Omron Sysmac Studio project 15-510_8110_20151007_10 (Sysmac Studio 1.1.4.95, StandardProject)

# Controller S8130_8140: NJ101-1000 version 1.10
Task PrimaryTask (priority 4, period or condition 1000): Program0, Program1, Program2, prS8120CCD

TYPE WORD_UNION : UNION
    Word_Type : WORD;
    Byte_Type : ARRAY[0..1] OF BYTE;
    Bool_Type : ARRAY[0..15] OF BOOL;
END_UNION END_TYPE
TYPE WorkType : STRUCT
    CCDSectionNo : INT;
    MotionData : Postion;
    QuantityofScrew : ARRAY[0..2] OF ScrewQuantity;
END_STRUCT END_TYPE
TYPE Postion : STRUCT
    Address : DINT;
    Speed : DINT;
END_STRUCT END_TYPE
TYPE ScrewQuantity : STRUCT
    Quantity : INT;
    ScrewJobNo : INT;
END_STRUCT END_TYPE
TYPE RecordData : STRUCT
    WorkingFlag : BOOL;
    FinishFlag : BOOL;
    OKFlag : BOOL;
    NGFlag : BOOL;
END_STRUCT END_TYPE
TYPE FH_CommandCode : (ChangeType := 3149824); END_TYPE

VAR_GLOBAL
    Reset_PB : BOOL;  (* 復歸開關; at IOBus://rack#0/slot#0/Ch1_In/Ch1_In00 *)
    EStop_PB : BOOL;  (* 急停開關; at IOBus://rack#0/slot#0/Ch1_In/Ch1_In01 *)
    CCDStart_PB : BOOL;  (* CCD啟動開關; at IOBus://rack#0/slot#0/Ch1_In/Ch1_In02 *)
    NGReject_SNR : BOOL;  (* 不良品排除檢測; at IOBus://rack#0/slot#0/Ch1_In/Ch1_In03 *)
    S8120_OK : BOOL;  (* at IOBus://rack#0/slot#0/Ch1_In/Ch1_In04 *)
    S8120_NG : BOOL;  (* at IOBus://rack#0/slot#0/Ch1_In/Ch1_In05 *)
    ASDA_IN_SRDY : BOOL;  (* at IOBus://rack#0/slot#0/Ch1_In/Ch1_In06 *)
    ASDA_IN_ZSPD : BOOL;  (* at IOBus://rack#0/slot#0/Ch1_In/Ch1_In07 *)
    ASDA_IN_HOME : BOOL;  (* at IOBus://rack#0/slot#0/Ch1_In/Ch1_In08 *)
    FeedScrew1_FeedSol : BOOL;  (* 送螺絲節流電磁閥1; at IOBus://rack#0/slot#0/Ch1_In/Ch1_In10 *)
    FeedScrew1_FeedSNR : BOOL;  (* 送螺絲螺絲檢知1; at IOBus://rack#0/slot#0/Ch1_In/Ch1_In11 *)
    FeedScrew2_FeedSol : BOOL;  (* 送螺絲節流電磁閥2; at IOBus://rack#0/slot#0/Ch1_In/Ch1_In12 *)
    FeedScrew2_FeedSNR : BOOL;  (* 送螺絲螺絲檢知2; at IOBus://rack#0/slot#0/Ch1_In/Ch1_In13 *)
    FeedScrew3_FeedSol : BOOL;  (* 送螺絲節流電磁閥3; at IOBus://rack#0/slot#0/Ch1_In/Ch1_In14 *)
    FeedScrew3_FeedSNR : BOOL;  (* 送螺絲螺絲檢知3; at IOBus://rack#0/slot#0/Ch1_In/Ch1_In15 *)
    Stanley1_IN_InCycle : BOOL;  (* 鎖付伺服左; at IOBus://rack#0/slot#0/Ch2_In/Ch2_In00 *)
    Stanley1_IN_Ready : BOOL;  (* 鎖付伺服左; at IOBus://rack#0/slot#0/Ch2_In/Ch2_In01 *)
    Stanley1_IN_DisassemblyDetected : BOOL;  (* 鎖付伺服左; at IOBus://rack#0/slot#0/Ch2_In/Ch2_In02 *)
    Stanley1_IN_JobSelectedBit0 : BOOL;  (* 鎖付伺服左; at IOBus://rack#0/slot#0/Ch2_In/Ch2_In03 *)
    Stanley1_IN_JobSelectedBit1 : BOOL;  (* 鎖付伺服左; at IOBus://rack#0/slot#0/Ch2_In/Ch2_In04 *)
    Stanley1_IN_JobSelectedBit2 : BOOL;  (* 鎖付伺服左; at IOBus://rack#0/slot#0/Ch2_In/Ch2_In05 *)
    Stanley1_IN_CycleOK : BOOL;  (* 鎖付伺服左; at IOBus://rack#0/slot#0/Ch2_In/Ch2_In06 *)
    Stanley1_IN_CycleNOK : BOOL;  (* 鎖付伺服左; at IOBus://rack#0/slot#0/Ch2_In/Ch2_In07 *)
    Stanley2_IN_InCycle : BOOL;  (* 鎖付伺服右; at IOBus://rack#0/slot#0/Ch2_In/Ch2_In08 *)
    Stanley2_IN_Ready : BOOL;  (* 鎖付伺服右; at IOBus://rack#0/slot#0/Ch2_In/Ch2_In09 *)
    Stanley2_IN_DisassemblyDetected : BOOL;  (* 鎖付伺服右; at IOBus://rack#0/slot#0/Ch2_In/Ch2_In10 *)
    Stanley2_IN_JobSelectedBit0 : BOOL;  (* 鎖付伺服右; at IOBus://rack#0/slot#0/Ch2_In/Ch2_In11 *)
    Stanley2_IN_JobSelectedBit1 : BOOL;  (* 鎖付伺服右; at IOBus://rack#0/slot#0/Ch2_In/Ch2_In12 *)
    Stanley2_IN_JobSelectedBit2 : BOOL;  (* 鎖付伺服右; at IOBus://rack#0/slot#0/Ch2_In/Ch2_In13 *)
    Stanley2_IN_CycleOK : BOOL;  (* 鎖付伺服右; at IOBus://rack#0/slot#0/Ch2_In/Ch2_In14 *)
    Stanley2_IN_CycleNOK : BOOL;  (* 鎖付伺服右; at IOBus://rack#0/slot#0/Ch2_In/Ch2_In15 *)
    FeedScrew1_FeedRY : BOOL;  (* 送螺絲啟動_1; at IOBus://rack#0/slot#1/Ch1_Out/Ch1_Out00 *)
    FeedScrew2_FeedRY : BOOL;  (* 送螺絲啟動_2; at IOBus://rack#0/slot#1/Ch1_Out/Ch1_Out01 *)
    FeedScrew3_FeedRY : BOOL;  (* 送螺絲啟動_3; at IOBus://rack#0/slot#1/Ch1_Out/Ch1_Out02 *)
    BZ : BOOL;  (* 蜂鳴器; at IOBus://rack#0/slot#1/Ch1_Out/Ch1_Out04 *)
    YL : BOOL;  (* 黃燈; at IOBus://rack#0/slot#1/Ch1_Out/Ch1_Out05 *)
    GL : BOOL;  (* 綠燈; at IOBus://rack#0/slot#1/Ch1_Out/Ch1_Out06 *)
    RL : BOOL;  (* 紅燈; at IOBus://rack#0/slot#1/Ch1_Out/Ch1_Out07 *)
    ASDA_OUT_ARST : BOOL;  (* at IOBus://rack#0/slot#1/Ch1_Out/Ch1_Out11 *)
    Stanley1_OUT_Start : BOOL;  (* 鎖付伺服左; at IOBus://rack#0/slot#1/Ch2_Out/Ch2_Out00 *)
    Stanley1_OUT_Stop : BOOL;  (* 鎖付伺服左; at IOBus://rack#0/slot#1/Ch2_Out/Ch2_Out01 *)
    Stanley1_OUT_Reverse : BOOL;  (* 鎖付伺服左; at IOBus://rack#0/slot#1/Ch2_Out/Ch2_Out02 *)
    Stanley1_OUT_JobBit0 : BOOL;  (* 鎖付伺服左; at IOBus://rack#0/slot#1/Ch2_Out/Ch2_Out03 *)
    Stanley1_OUT_JobBit1 : BOOL;  (* 鎖付伺服左; at IOBus://rack#0/slot#1/Ch2_Out/Ch2_Out04 *)
    Stanley1_OUT_JobBit2 : BOOL;  (* 鎖付伺服左; at IOBus://rack#0/slot#1/Ch2_Out/Ch2_Out05 *)
    Stanley1_OUT_RsetJob : BOOL;  (* 鎖付伺服左; at IOBus://rack#0/slot#1/Ch2_Out/Ch2_Out06 *)
    Stanley1_OUT_Ignored : BOOL;  (* 鎖付伺服左; at IOBus://rack#0/slot#1/Ch2_Out/Ch2_Out07 *)
    Stanley2_OUT_Start : BOOL;  (* 鎖付伺服右; at IOBus://rack#0/slot#1/Ch2_Out/Ch2_Out08 *)
    Stanley2_OUT_Stop : BOOL;  (* 鎖付伺服右; at IOBus://rack#0/slot#1/Ch2_Out/Ch2_Out09 *)
    Stanley2_OUT_Reverse : BOOL;  (* 鎖付伺服右; at IOBus://rack#0/slot#1/Ch2_Out/Ch2_Out10 *)
    Stanley2_OUT_JobBit0 : BOOL;  (* 鎖付伺服右; at IOBus://rack#0/slot#1/Ch2_Out/Ch2_Out11 *)
    Stanley2_OUT_JobBit1 : BOOL;  (* 鎖付伺服右; at IOBus://rack#0/slot#1/Ch2_Out/Ch2_Out12 *)
    Stanley2_OUT_JobBit2 : BOOL;  (* 鎖付伺服右; at IOBus://rack#0/slot#1/Ch2_Out/Ch2_Out13 *)
    Stanley2_OUT_RsetJob : BOOL;  (* 鎖付伺服右; at IOBus://rack#0/slot#1/Ch2_Out/Ch2_Out14 *)
    Stanley2_OUT_Ignored : BOOL;  (* 鎖付伺服右; at IOBus://rack#0/slot#1/Ch2_Out/Ch2_Out15 *)
    E002_Line0_Command_Request : BOOL;  (* at ECAT://node#1/Line0 Command Request *)
    CCD1_Trigger : BOOL;  (* CCD1; at ECAT://node#1/Line0 Trigger *)
    CCD1_Error_Clear : BOOL;  (* CCD1; at ECAT://node#1/Line0 Error Clear *)
    E002_Line0_Command_Code : DWORD;  (* at ECAT://node#1/Line0 Command Code *)
    E002_Line0_Command_Parameter_0 : DINT;  (* at ECAT://node#1/Line0 Command Parameter 0 *)
    E002_Line0_Command_Completion : BOOL;  (* at ECAT://node#1/Line0 Command Completion *)
    CCD1_Busy : BOOL;  (* CCD1; at ECAT://node#1/Line0 Busy *)
    CCD1_Trigger_Ready : BOOL;  (* CCD1; at ECAT://node#1/Line0 Trigger Ready *)
    E002_Line0_Run_Mode : BOOL;  (* at ECAT://node#1/Line0 Run Mode *)
    E002_Line0_Trigger_Ack : BOOL;  (* at ECAT://node#1/Line0 Trigger Ack *)
    E002_Line0_Command_Ready : BOOL;  (* at ECAT://node#1/Line0 Command Ready *)
    CCD1_ResultData0 : DINT;  (* at ECAT://node#1/Line0 DINT Result Data 0 *)
    CCD1_ResultData1 : DINT;  (* at ECAT://node#1/Line0 DINT Result Data 1 *)
    E002_Line1_Command_Request : BOOL;  (* at ECAT://node#1/Line1 Command Request *)
    CCD2_Trigger : BOOL;  (* CCD2; at ECAT://node#1/Line1 Trigger *)
    CCD2_Error_Clear : BOOL;  (* CCD2; at ECAT://node#1/Line1 Error Clear *)
    E002_Line1_Command_Code : DWORD;  (* at ECAT://node#1/Line1 Command Code *)
    E002_Line1_Command_Parameter_0 : DINT;  (* at ECAT://node#1/Line1 Command Parameter 0 *)
    E002_Line1_Command_Completion : BOOL;  (* at ECAT://node#1/Line1 Command Completion *)
    CCD2_Busy : BOOL;  (* CCD2; at ECAT://node#1/Line1 Busy *)
    CCD2_Trigger_Ready : BOOL;  (* CCD2; at ECAT://node#1/Line1 Trigger Ready *)
    E002_Line1_Run_Mode : BOOL;  (* at ECAT://node#1/Line1 Run Mode *)
    E002_Line1_Command_Ready : BOOL;  (* at ECAT://node#1/Line1 Command Ready *)
    CCD2_ResultData0 : DINT;  (* at ECAT://node#1/Line1 DINT Result Data 0 *)
    CCD2_ResultData1 : DINT;  (* at ECAT://node#1/Line1 DINT Result Data 1 *)
    FeedStartFlag_1 : BOOL;
    FeedStartFlag_2 : BOOL;
    FeedStartFlag_3 : BOOL;
    Go_Home_Auto : BOOL;
    Go_Zero_Auto : BOOL;
    Go_Position_Auto : BOOL;
    CCD1_Triger_Auto : BOOL;
    CCD2_Triger_Auto : BOOL;
    CCD1_Finish_Flag : BOOL;
END_VAR
VAR_GLOBAL RETAIN
    TypeNo AT %D0 : ARRAY[0..7] OF WorkType;  (* published *)
    HMI_CurrentWorkType AT %D500 : INT;  (* published *)
    HMI_CurrentFeedScrewQuantity_8110 AT %D1000 : INT;  (* 送出的螺絲計數; published *)
    HMI_CurrentFeedScrewQuantity_8130 AT %D1001 : INT;  (* 送出的螺絲計數; published *)
    HMI_CurrentFeedScrewQuantity_8140 AT %D1002 : INT;  (* 送出的螺絲計數; published *)
    HMI_CurrentScrewQuantity_8110 AT %D1003 : INT;  (* 已鎖的螺絲計數; published *)
    HMI_CurrentScrewQuantity_8130 AT %D1004 : INT;  (* 已鎖的螺絲計數; published *)
    HMI_CurrentScrewQuantity_8140 AT %D1005 : INT;  (* 已鎖的螺絲計數; published *)
    HMI_CurrentAddress AT %D1006 : DINT;  (* 目前位置; published *)
    HMI_CurrentSpeed AT %D1008 : DINT;  (* 目前速度; published *)
    RejectPosition_Address AT %D1010 : DINT;  (* CCD退料位置; published *)
    Error_FeedScrew1_FeedSNR AT %D3000.0 : BOOL;  (* published *)
    Error_FeedScrew2_FeedSNR AT %D3000.1 : BOOL;  (* published *)
    Error_FeedScrew3_FeedSNR AT %D3000.2 : BOOL;  (* published *)
    Error_CCDTrigOver3Times AT %D3000.3 : BOOL;  (* published *)
    Error_Over1timeECatError AT %D3000.4 : BOOL;  (* published *)
    Error_EtherNetError AT %D3000.5 : BOOL;  (* published *)
    Error_Stanley1_Ready AT %D3000.6 : BOOL;  (* published *)
    Error_Stanley2_Ready AT %D3000.7 : BOOL;  (* published *)
    Error_Servo_Ready AT %D3000.8 : BOOL;  (* published *)
    Error_EStop_PB AT %D3000.9 : BOOL;  (* published *)
    Error_CCD1_Ready AT %D3000.10 : BOOL;  (* published *)
    Error_CCD2_Ready AT %D3000.11 : BOOL;  (* published *)
END_VAR
VAR_GLOBAL
    StationData AT %W0 : ARRAY[0..3] OF RecordData;  (* published *)
END_VAR
VAR_GLOBAL RETAIN
    HMI_FeedScrewPB_1 AT %H100.0 : BOOL;  (* published *)
    HMI_FeedScrewPB_2 AT %H101.0 : BOOL;  (* published *)
    HMI_FeedScrewPB_3 AT %H102.0 : BOOL;  (* published *)
    HMI_AutoStartPB AT %H103.0 : BOOL;  (* published *)
    HMI_MachineRunStatus AT %H104.0 : BOOL;  (* published *)
    HMI_PandingOKPB AT %H105.0 : BOOL;  (* published *)
    HMI_AutoStatus AT %H106.0 : BOOL;  (* published *)
    HMI_ManualStatus AT %H107.0 : BOOL;  (* published *)
    HMI_BZ_Status AT %H108.0 : BOOL;  (* published *)
    HMI_CCD1PB AT %H109.0 : BOOL;  (* published *)
    HMI_PandingNGPB AT %H110.0 : BOOL;  (* published *)
    HMI_AutoStartPB_Continum AT %H111.0 : BOOL;  (* published *)
    NGStatus AT %H112.0 : BOOL;  (* published *)
    Go_Home AT %H113.0 : BOOL;  (* published *)
    Go_Zero AT %H114.0 : BOOL;  (* published *)
    Go_Postion AT %H115.0 : BOOL;  (* published *)
    HMI_CCD_OK AT %H116.0 : BOOL;  (* published *)
    HMI_CCD_NG AT %H117.0 : BOOL;  (* published *)
    HMI_S8120_OK AT %H118.0 : BOOL;  (* published *)
    HMI_S8120_NG AT %H119.0 : BOOL;  (* published *)
    HMI_NGReject_PB AT %H120.0 : BOOL;  (* published *)
    HMI_Start8110_PB AT %H121.0 : BOOL;  (* published *)
    HMI_Start8130_PB AT %H122.0 : BOOL;  (* published *)
    HMI_Start8140_PB AT %H123.0 : BOOL;  (* published *)
    HMI_Manual_PB AT %H124.0 : BOOL;  (* published *)
    Go_Position_Reject AT %H125.0 : BOOL;  (* published *)
    CCDSectionChangeFlag AT %H126.0 : BOOL;  (* published *)
    GoHomedFlag AT %H127.0 : BOOL;  (* published *)
    CCDSettingFlag AT %H128.0 : BOOL;  (* published *)
    HMI_8120CCDBackPB AT %H130.0 : BOOL;  (* published *)
    HMI_8120CCDOutPB AT %H131.0 : BOOL;  (* published *)
    HMI_8120STARTPB AT %H132.0 : BOOL;  (* published *)
    HMI_8120CCDstartPB AT %H133.0 : BOOL;  (* published *)
    FQ2_NG AT %H134.0 : BOOL;  (* published *)
    FQ2_Busy AT %H135.0 : BOOL;  (* published *)
END_VAR
VAR_GLOBAL
    ResetPB_8190 : BOOL;  (* 8190復歸按鍵; network input *)
    CCDStartFlag_8190 : BOOL;  (* 8190CCD啟動; network input *)
    CCDStartPB_8190 : BOOL;  (* 8190CCD啟動手動按鍵; network input *)
    CCDCheckOK_8190 : BOOL;  (* 8190檢查OK; network output *)
    CCDCheckNG_8190 : BOOL;  (* 8190檢查NG; network output *)
    CCDOver3TimesError_8190 : BOOL;  (* 8190超過三次CCD沒回應; network output *)
    CCDSectionChange : BOOL;  (* network input *)
    CCDSectionNo : INT;  (* network input *)
    CCDSectionChangeComplete : BOOL;  (* network output *)
    S8140OK : BOOL;  (* network output *)
    S8140NG : BOOL;  (* network output *)
    Mapping_Controlword_6040_00 : WORD_UNION;
    Mapping_Statusword_6041_00 : WORD_UNION;
    E001_1st_RxPDO_Mapping_Controlword_6040_00 : UINT;  (* at ECAT://node#5/1st RxPDO Mapping_Controlword_6040_00 *)
    E001_1st_RxPDO_Mapping_Modes_of_operation_6060_00 : SINT;  (* at ECAT://node#5/1st RxPDO Mapping_Modes of operation_6060_00 *)
    E001_1st_RxPDO_Mapping_Target_position_607A_00 : DINT;  (* at ECAT://node#5/1st RxPDO Mapping_Target position_607A_00 *)
    E001_1st_RxPDO_Mapping_Profile_velocity_6081_00 : UDINT;  (* at ECAT://node#5/1st RxPDO Mapping_Profile velocity_6081_00 *)
    E001_1st_RxPDO_Mapping_Homing_method_6098_00 : SINT;  (* at ECAT://node#5/1st RxPDO Mapping_Homing method_6098_00 *)
    E001_1st_RxPDO_Mapping_Home_offset_607C_00 : DINT;
    E001_1st_TxPDO_Mapping_Statusword_6041_00 : UINT;  (* at ECAT://node#5/1st TxPDO Mapping_Statusword_6041_00 *)
    E001_1st_TxPDO_Mapping_Position_actual_value_6064_00 : DINT;  (* at ECAT://node#5/1st TxPDO Mapping_Position actual value_6064_00 *)
    E001_1st_TxPDO_Mapping_Velocity_actual_value_606C_00 : DINT;  (* at ECAT://node#5/1st TxPDO Mapping_Velocity actual value_606C_00 *)
    E001_1st_RxPDO_Mapping_Profile_acceleration_6083_00 : UDINT;  (* at ECAT://node#5/1st RxPDO Mapping_Profile acceleration_6083_00 *)
    E001_1st_RxPDO_Mapping_Profile_deceleration_6084_00 : UDINT;  (* at ECAT://node#5/1st RxPDO Mapping_Profile deceleration_6084_00 *)
    E001_1st_RxPDO_Mapping_Speed_during_search_for_swi_6099_01 : UDINT;  (* at ECAT://node#5/1st RxPDO Mapping_Speed during search for swi_6099_01 *)
    Check8120Back_SOL : BOOL;  (* CCD檢查氣缸歸SOL; at IOBus://rack#0/slot#3/Ch1_Out/Ch1_Out00 *)
    Check8120Out_SOL : BOOL;  (* CCD檢查氣缸出SOL; at IOBus://rack#0/slot#3/Ch1_Out/Ch1_Out01 *)
    Check8120Back_LS : BOOL;  (* CCD檢查氣缸歸LS; at IOBus://rack#0/slot#2/Ch1_In/Ch1_In00 *)
    Check8120Out_LS : BOOL;  (* CCD檢查氣缸出LS; at IOBus://rack#0/slot#2/Ch1_In/Ch1_In01 *)
    Check8120_CCDNG : BOOL;  (* FQ2NG訊號; at IOBus://rack#0/slot#2/Ch1_In/Ch1_In02 *)
    Check8120_CCDBusy : BOOL;  (* FQ2Busy訊號; at IOBus://rack#0/slot#2/Ch1_In/Ch1_In03 *)
    Check8120_CCDIN0 : BOOL;  (* FQ2埸景bit0; at IOBus://rack#0/slot#3/Ch1_Out/Ch1_Out02 *)
    Check8120_CCDIN1 : BOOL;  (* FQ2埸景bit1; at IOBus://rack#0/slot#3/Ch1_Out/Ch1_Out03 *)
    Check8120_CCDIN2 : BOOL;  (* FQ2埸景bit2; at IOBus://rack#0/slot#3/Ch1_Out/Ch1_Out04 *)
    Check8120_CCDIN3 : BOOL;  (* FQ2埸景bit3; at IOBus://rack#0/slot#3/Ch1_Out/Ch1_Out05 *)
    Check8120_CCDIN4 : BOOL;  (* FQ2埸景bit4; at IOBus://rack#0/slot#3/Ch1_Out/Ch1_Out06 *)
    Check8120_CCDIN5 : BOOL;  (* FQ2埸景bit5; at IOBus://rack#0/slot#3/Ch1_Out/Ch1_Out07 *)
    Check8120_CCDTrig : BOOL;  (* FQ2CCDTrigger訊號; at IOBus://rack#0/slot#3/Ch1_Out/Ch1_Out08 *)
    Check8120_CCDStartPB : BOOL;  (* S8120CCD起動按鍵; at IOBus://rack#0/slot#2/Ch1_In/Ch1_In04 *)
    CCD0CheckOK : BOOL;
    CCD0CheckNG : BOOL;
END_VAR

PROGRAM Program0
VAR
    TON_BZ : TON;
    M8013 : BOOL;
    TON_BZON : TON;
    TON_StopBZ : TON;
    FeedScrewFlow_8110 : FeedScrewFlow;
    FeedScrewFlow_8130 : FeedScrewFlow;
    FeedScrewFlow_8140 : FeedScrewFlow;
    Screw_8110 : StanleyScrewFlow;
    Screw_8130 : StanleyScrewFlow;
    Screw_8140 : StanleyScrewFlow;
    JobSelect_8110 : StanleyJobSelect;
    JobSelect_8130 : StanleyJobSelect;
    JobSelect_8140 : StanleyJobSelect;
    CCD_Line0 : CCD;
    CCD_Line１ : CCD;
    ccd1 : BOOL;
    ECErrorReset : ResetECError;
    PowerOn : BOOL;
    Idle : BOOL;
    Ton_PON : TON;
    MainProgram_8110 : Station_2Step;
    MainProgram_8130 : Station_2Step;
    MainProgram_8140 : Station_2Step;
    Step1StartFlag_8110 : BOOL;  (* 送螺絲開始 *)
    Step1StartFlag_8130 : BOOL;  (* 送螺絲開始 *)
    Step1StartFlag_8140 : BOOL;  (* 送螺絲開始 *)
    Step1FinishFlag_8110 : BOOL;  (* 送螺絲完成 *)
    Step1FinishFlag_8130 : BOOL;  (* 送螺絲完成 *)
    Step1FinishFlag_8140 : BOOL;  (* 送螺絲完成 *)
    Step2StartFlag_8110 : BOOL;  (* 鎖螺絲開始 *)
    Step2StartFlag_8140 : BOOL;  (* 鎖螺絲開始 *)
    ScrewOKFlag_8110 : BOOL;
    ScrewNGFlag_8110 : BOOL;
    ScrewOKFlag_8130 : BOOL;
    ScrewNGFlag_8130 : BOOL;
    ScrewOKFlag_8140 : BOOL;
    ScrewNGFlag_8140 : BOOL;
    DataNGStatus : BOOL;
    FeedScrewNGStatus : BOOL;
    ECatErrorCounter : INT;
    Error_EtherCatError : BOOL;
    TON_POWERON : TON;
    FlowStart_8130 : BOOL;
    Step2StartFlag_8130 : BOOL;
    jobbit0_8130 : BOOL;
    jobbit1_8130 : BOOL;
    jobbit2_8130 : BOOL;
    jobbit0_8140 : BOOL;
    jobbit1_8140 : BOOL;
    jobbit2_8140 : BOOL;
    MachineStartStatus : BOOL;
    NGStartFlag : BOOL;
    ton_ngstart : TON;
    Start8110 : BOOL;
    Start8130 : BOOL;
    Start8140 : BOOL;
END_VAR
VAR_EXTERNAL
    Error_FeedScrew1_FeedSNR : BOOL;
    Error_FeedScrew2_FeedSNR : BOOL;
    Error_FeedScrew3_FeedSNR : BOOL;
    BZ : BOOL;
    YL : BOOL;
    GL : BOOL;
    RL : BOOL;
    HMI_MachineRunStatus : BOOL;
    HMI_BZ_Status : BOOL;
    HMI_AutoStartPB : BOOL;  (* 人機起動按鍵 *)
    FeedScrew1_FeedSol : BOOL;
    HMI_CurrentWorkType : INT;
    TypeNo : ARRAY[0..7] OF WorkType;
    HMI_CurrentFeedScrewQuantity_8110 : INT;
    FeedScrew1_FeedRY : BOOL;
    FeedStartFlag_1 : BOOL;
    Stanley1_IN_CycleNOK : BOOL;
    Stanley1_IN_CycleOK : BOOL;
    Stanley1_IN_InCycle : BOOL;
    StationData : ARRAY[0..3] OF RecordData;
    FeedStartFlag_2 : BOOL;
    FeedScrew2_FeedSol : BOOL;
    FeedScrew3_FeedSol : BOOL;
    HMI_CurrentFeedScrewQuantity_8130 : INT;
    FeedStartFlag_3 : BOOL;
    Stanley2_IN_CycleNOK : BOOL;
    Stanley2_IN_CycleOK : BOOL;
    Stanley2_IN_InCycle : BOOL;
    Stanley1_OUT_JobBit0 : BOOL;
    Stanley1_OUT_JobBit1 : BOOL;
    Stanley1_OUT_JobBit2 : BOOL;
    Stanley2_OUT_JobBit0 : BOOL;
    Stanley2_OUT_JobBit1 : BOOL;
    Stanley2_OUT_JobBit2 : BOOL;
    CCD1_Trigger : BOOL;
    HMI_CCD1PB : BOOL;
    Reset_PB : BOOL;
    CCD1_ResultData0 : DINT;
    CCD1_ResultData1 : DINT;
    Error_CCDTrigOver3Times : BOOL;
    ResetPB_8190 : BOOL;
    CCDStartFlag_8190 : BOOL;
    CCDStartPB_8190 : BOOL;
    CCDCheckOK_8190 : BOOL;
    CCDCheckNG_8190 : BOOL;
    CCD2_Trigger : BOOL;
    CCDOver3TimesError_8190 : BOOL;
    CCD1_Trigger_Ready : BOOL;
    CCD2_Trigger_Ready : BOOL;
    Error_EtherNetError : BOOL;
    HMI_PandingOKPB : BOOL;
    HMI_PandingNGPB : BOOL;
    Stanley1_IN_Ready : BOOL;
    Stanley2_IN_Ready : BOOL;
    Error_Stanley1_Ready : BOOL;
    Error_Stanley2_Ready : BOOL;
    HMI_AutoStartPB_Continum : BOOL;
    NGReject_SNR : BOOL;
    Error_Over1timeECatError : BOOL;
    HMI_CurrentScrewQuantity_8110 : INT;
    HMI_CurrentScrewQuantity_8140 : INT;
    HMI_CurrentFeedScrewQuantity_8140 : INT;
    NGStatus : BOOL;
    S8120_OK : BOOL;
    Stanley2_IN_JobSelectedBit0 : BOOL;
    Stanley2_IN_JobSelectedBit1 : BOOL;
    Stanley2_IN_JobSelectedBit2 : BOOL;
    HMI_CurrentScrewQuantity_8130 : INT;
    HMI_CCD_NG : BOOL;
    HMI_CCD_OK : BOOL;
    CCD1_Triger_Auto : BOOL;
    CCD1_Finish_Flag : BOOL;
    HMI_S8120_OK : BOOL;
    S8120_NG : BOOL;
    HMI_S8120_NG : BOOL;
    HMI_NGReject_PB : BOOL;
    ASDA_IN_SRDY : BOOL;
    Error_Servo_Ready : BOOL;
    EStop_PB : BOOL;
    Error_EStop_PB : BOOL;
    Error_CCD1_Ready : BOOL;
    Error_CCD2_Ready : BOOL;
    HMI_Start8110_PB : BOOL;
    HMI_Start8130_PB : BOOL;
    HMI_Start8140_PB : BOOL;
    HMI_Manual_PB : BOOL;
    CCD2_ResultData0 : DINT;
    CCD2_ResultData1 : DINT;
    CCDSettingFlag : BOOL;
    CCD0CheckOK : BOOL;
    CCD0CheckNG : BOOL;
    E002_Line0_Run_Mode : BOOL;
    E002_Line1_Run_Mode : BOOL;
    CCD1_Busy : BOOL;
    CCD2_Busy : BOOL;
END_VAR
VAR
    _e1 : R_TRIG;
    _e2 : R_TRIG;
    _e3 : R_TRIG;
    _e4 : R_TRIG;
    _e5 : R_TRIG;
    _e6 : F_TRIG;
    _e7 : R_TRIG;
    _e8 : R_TRIG;
    _e9 : R_TRIG;
    _e10 : R_TRIG;
    _e11 : R_TRIG;
    _e12 : R_TRIG;
    _e13 : R_TRIG;
    _e14 : F_TRIG;
END_VAR

(* Section Section_Main: ladder, written here as Structured Text *)

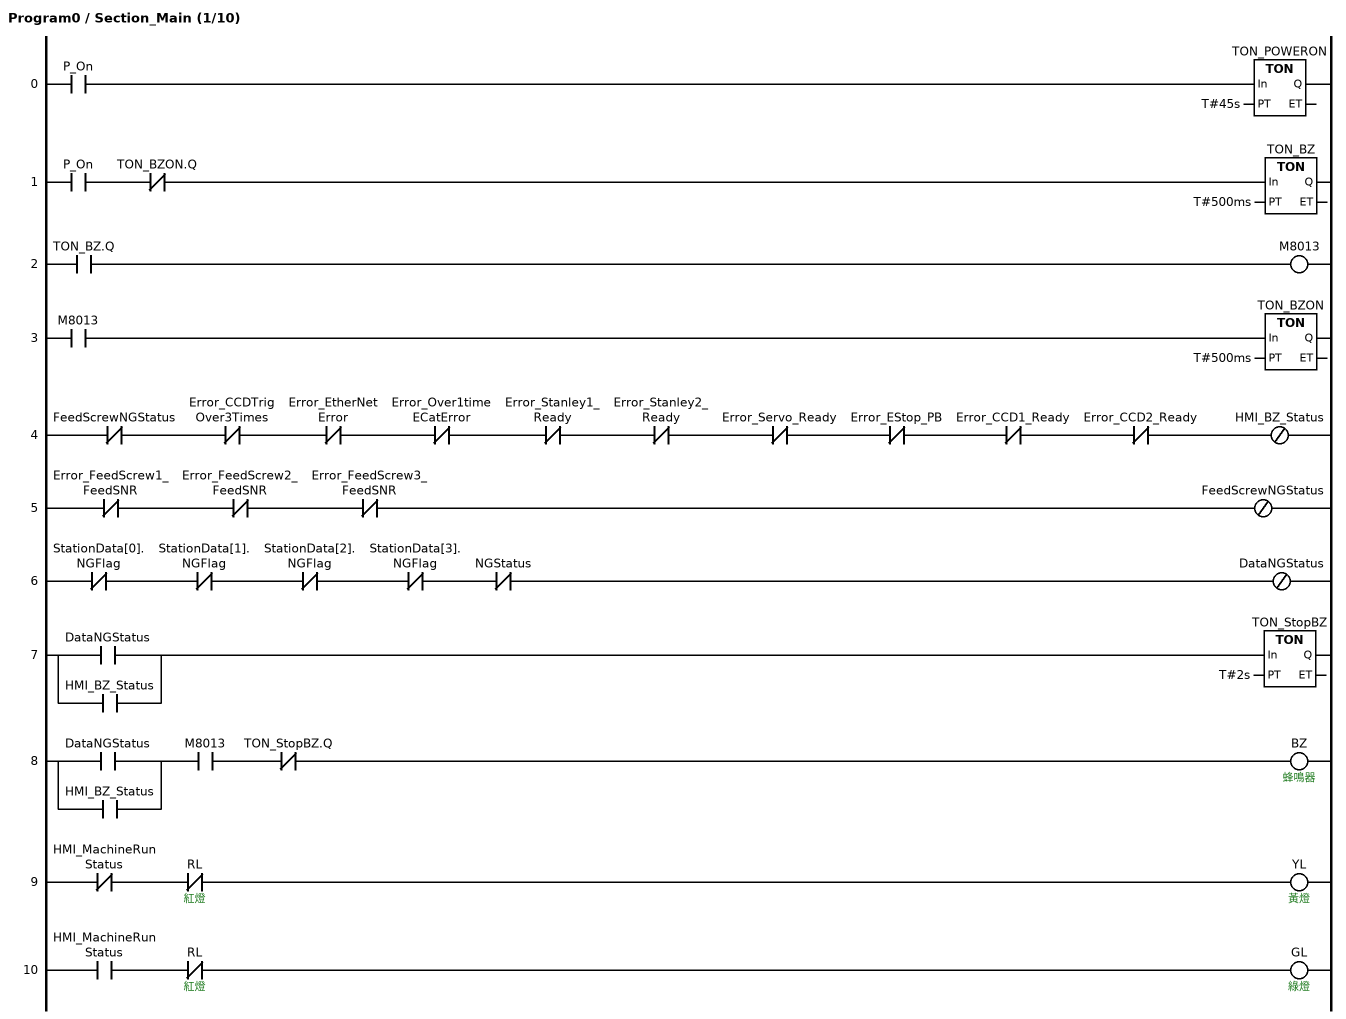
(* Rung 0 *)
TON_POWERON(In := P_On, PT := T#45s);
(* Rung 1 *)
TON_BZ(In := P_On AND NOT TON_BZON.Q, PT := T#500ms);
(* Rung 2 *)
M8013 := TON_BZ.Q;
(* Rung 3 *)
TON_BZON(In := M8013, PT := T#500ms);
(* Rung 4 *)
HMI_BZ_Status := NOT (NOT FeedScrewNGStatus AND NOT Error_CCDTrigOver3Times AND NOT Error_EtherNetError AND NOT Error_Over1timeECatError AND NOT Error_Stanley1_Ready AND NOT Error_Stanley2_Ready AND NOT Error_Servo_Ready AND NOT Error_EStop_PB AND NOT Error_CCD1_Ready AND NOT Error_CCD2_Ready);
(* Rung 5 *)
FeedScrewNGStatus := NOT (NOT Error_FeedScrew1_FeedSNR AND NOT Error_FeedScrew2_FeedSNR AND NOT Error_FeedScrew3_FeedSNR);
(* Rung 6 *)
DataNGStatus := NOT (NOT StationData[0].NGFlag AND NOT StationData[1].NGFlag AND NOT StationData[2].NGFlag AND NOT StationData[3].NGFlag AND NOT NGStatus);
(* Rung 7 *)
TON_StopBZ(In := DataNGStatus OR HMI_BZ_Status, PT := T#2s);
(* Rung 8 *)
BZ := (DataNGStatus OR HMI_BZ_Status) AND M8013 AND NOT TON_StopBZ.Q;
(* Rung 9 *)
YL := NOT HMI_MachineRunStatus AND NOT RL;
(* Rung 10 *)
GL := HMI_MachineRunStatus AND NOT RL;

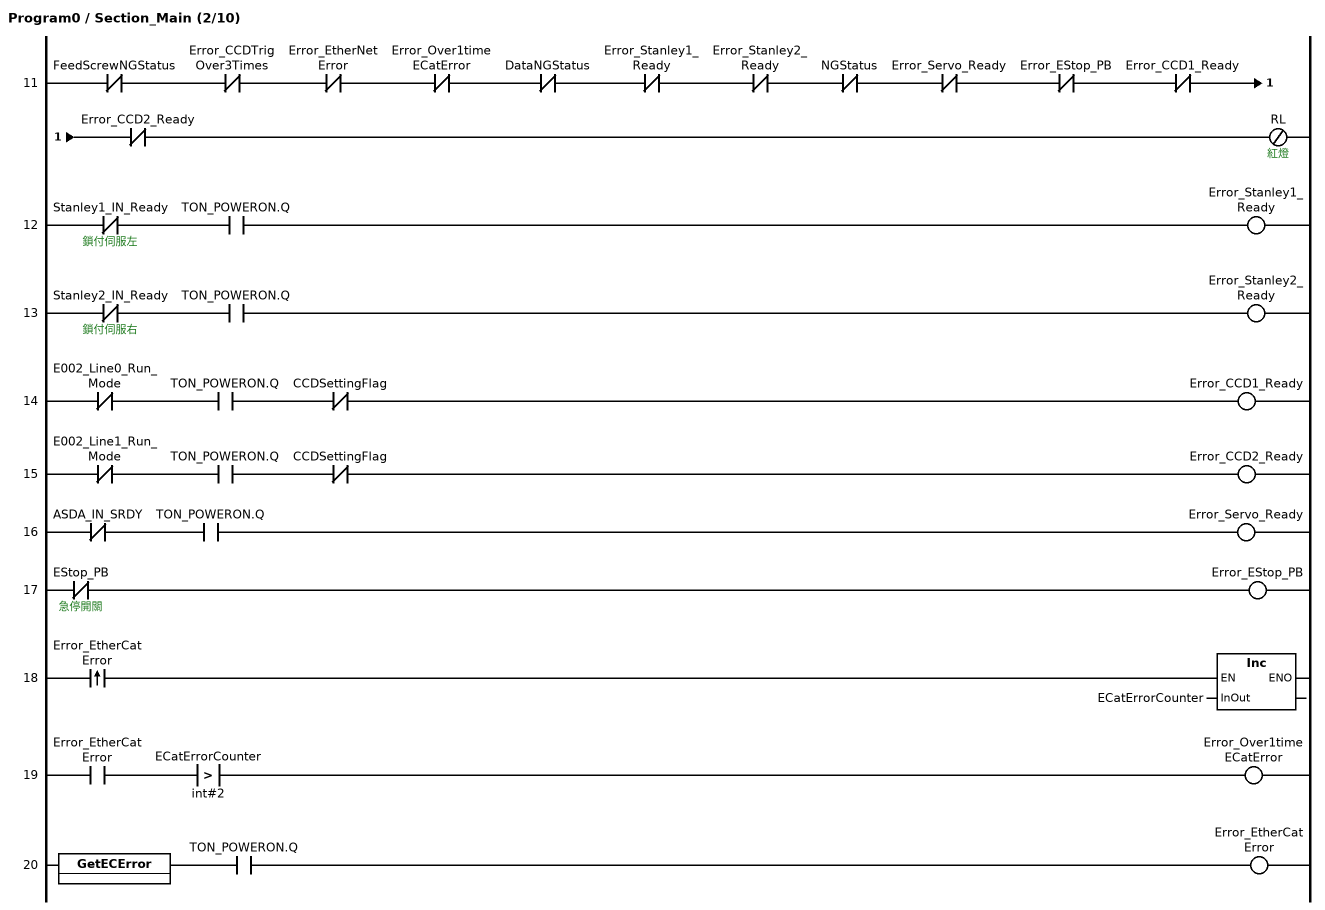
(* Rung 11 *)
RL := NOT (NOT FeedScrewNGStatus AND NOT Error_CCDTrigOver3Times AND NOT Error_EtherNetError AND NOT Error_Over1timeECatError AND NOT DataNGStatus AND NOT Error_Stanley1_Ready AND NOT Error_Stanley2_Ready AND NOT NGStatus AND NOT Error_Servo_Ready AND NOT Error_EStop_PB AND NOT Error_CCD1_Ready AND NOT Error_CCD2_Ready);
(* Rung 12 *)
Error_Stanley1_Ready := NOT Stanley1_IN_Ready AND TON_POWERON.Q;
(* Rung 13 *)
Error_Stanley2_Ready := NOT Stanley2_IN_Ready AND TON_POWERON.Q;
(* Rung 14 *)
Error_CCD1_Ready := NOT E002_Line0_Run_Mode AND TON_POWERON.Q AND NOT CCDSettingFlag;
(* Rung 15 *)
Error_CCD2_Ready := NOT E002_Line1_Run_Mode AND TON_POWERON.Q AND NOT CCDSettingFlag;
(* Rung 16 *)
Error_Servo_Ready := NOT ASDA_IN_SRDY AND TON_POWERON.Q;
(* Rung 17 *)
Error_EStop_PB := NOT EStop_PB;
(* Rung 18 *)
_e1(CLK := Error_EtherCatError);
IF _e1.Q THEN Inc(InOut := ECatErrorCounter); END_IF;
(* Rung 19 *)
Error_Over1timeECatError := Error_EtherCatError AND (ECatErrorCounter > int#2);
(* Rung 20 *)
Error_EtherCatError := GetECError() AND TON_POWERON.Q;

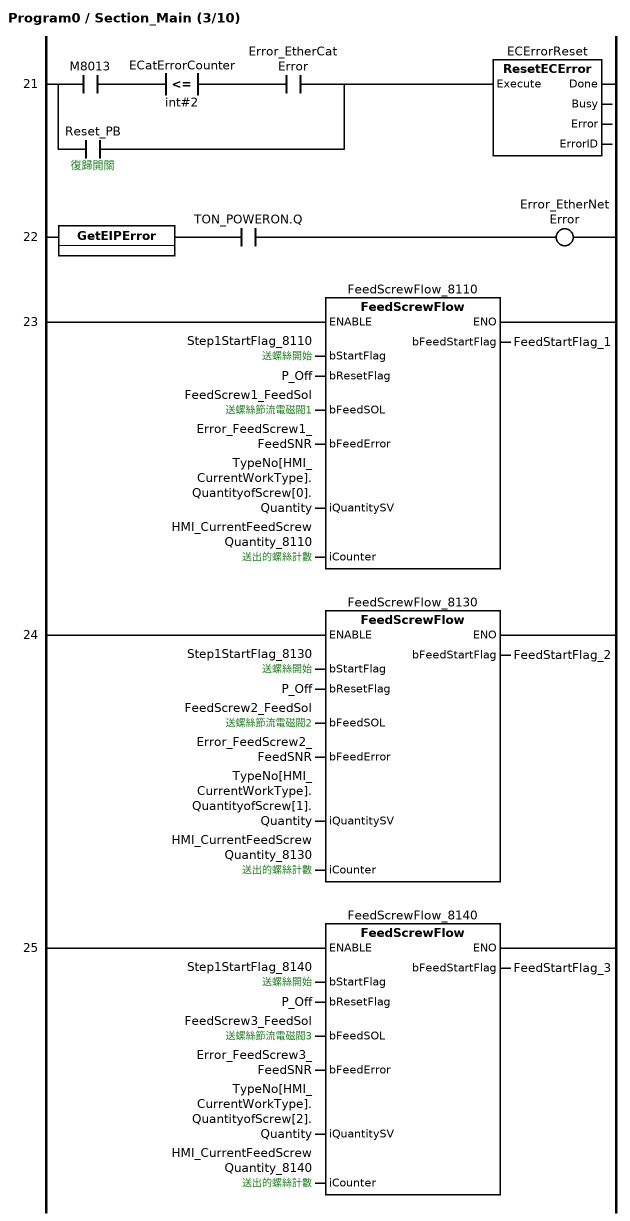
(* Rung 21 *)
ECErrorReset(Execute := (M8013 AND (ECatErrorCounter <= int#2) AND Error_EtherCatError) OR Reset_PB);
(* Rung 22 *)
Error_EtherNetError := GetEIPError() AND TON_POWERON.Q;
(* Rung 23 *)
FeedScrewFlow_8110(ENABLE := TRUE, bStartFlag := Step1StartFlag_8110, bResetFlag := P_Off, bFeedSOL := FeedScrew1_FeedSol, bFeedError := Error_FeedScrew1_FeedSNR, iQuantitySV := TypeNo[HMI_CurrentWorkType].QuantityofScrew[0].Quantity, iCounter := HMI_CurrentFeedScrewQuantity_8110, bFeedStartFlag => FeedStartFlag_1);
(* Rung 24 *)
FeedScrewFlow_8130(ENABLE := TRUE, bStartFlag := Step1StartFlag_8130, bResetFlag := P_Off, bFeedSOL := FeedScrew2_FeedSol, bFeedError := Error_FeedScrew2_FeedSNR, iQuantitySV := TypeNo[HMI_CurrentWorkType].QuantityofScrew[1].Quantity, iCounter := HMI_CurrentFeedScrewQuantity_8130, bFeedStartFlag => FeedStartFlag_2);
(* Rung 25 *)
FeedScrewFlow_8140(ENABLE := TRUE, bStartFlag := Step1StartFlag_8140, bResetFlag := P_Off, bFeedSOL := FeedScrew3_FeedSol, bFeedError := Error_FeedScrew3_FeedSNR, iQuantitySV := TypeNo[HMI_CurrentWorkType].QuantityofScrew[2].Quantity, iCounter := HMI_CurrentFeedScrewQuantity_8140, bFeedStartFlag => FeedStartFlag_3);

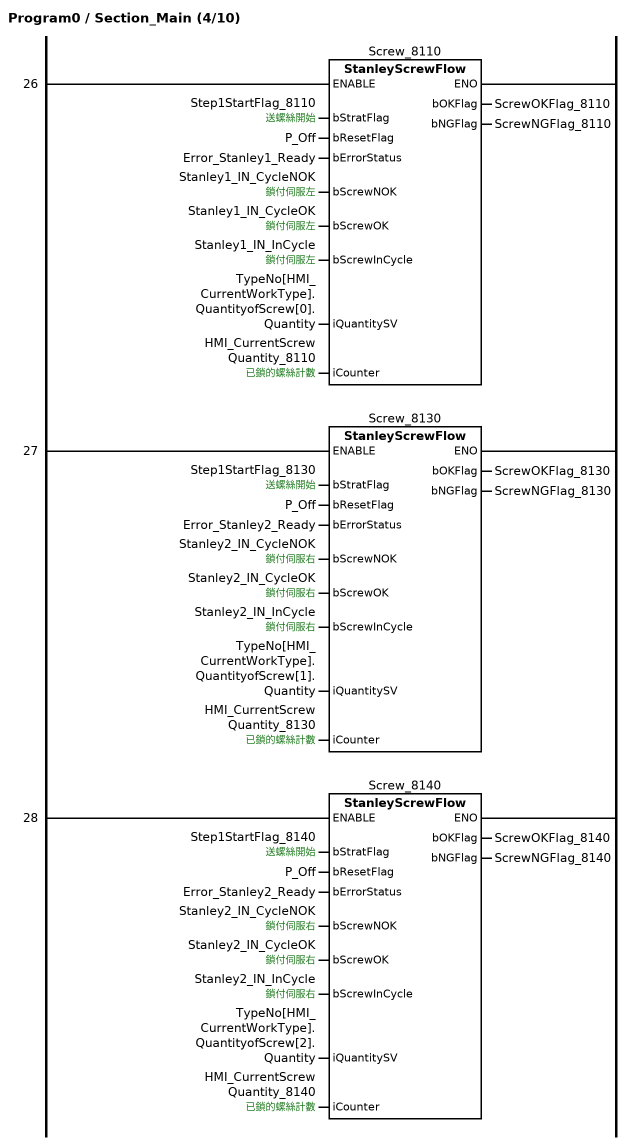
(* Rung 26 *)
Screw_8110(ENABLE := TRUE, bStratFlag := Step1StartFlag_8110, bResetFlag := P_Off, bErrorStatus := Error_Stanley1_Ready, bScrewNOK := Stanley1_IN_CycleNOK, bScrewOK := Stanley1_IN_CycleOK, bScrewInCycle := Stanley1_IN_InCycle, iQuantitySV := TypeNo[HMI_CurrentWorkType].QuantityofScrew[0].Quantity, iCounter := HMI_CurrentScrewQuantity_8110, bOKFlag => ScrewOKFlag_8110, bNGFlag => ScrewNGFlag_8110);
(* Rung 27 *)
Screw_8130(ENABLE := TRUE, bStratFlag := Step1StartFlag_8130, bResetFlag := P_Off, bErrorStatus := Error_Stanley2_Ready, bScrewNOK := Stanley2_IN_CycleNOK, bScrewOK := Stanley2_IN_CycleOK, bScrewInCycle := Stanley2_IN_InCycle, iQuantitySV := TypeNo[HMI_CurrentWorkType].QuantityofScrew[1].Quantity, iCounter := HMI_CurrentScrewQuantity_8130, bOKFlag => ScrewOKFlag_8130, bNGFlag => ScrewNGFlag_8130);
(* Rung 28 *)
Screw_8140(ENABLE := TRUE, bStratFlag := Step1StartFlag_8140, bResetFlag := P_Off, bErrorStatus := Error_Stanley2_Ready, bScrewNOK := Stanley2_IN_CycleNOK, bScrewOK := Stanley2_IN_CycleOK, bScrewInCycle := Stanley2_IN_InCycle, iQuantitySV := TypeNo[HMI_CurrentWorkType].QuantityofScrew[2].Quantity, iCounter := HMI_CurrentScrewQuantity_8140, bOKFlag => ScrewOKFlag_8140, bNGFlag => ScrewNGFlag_8140);

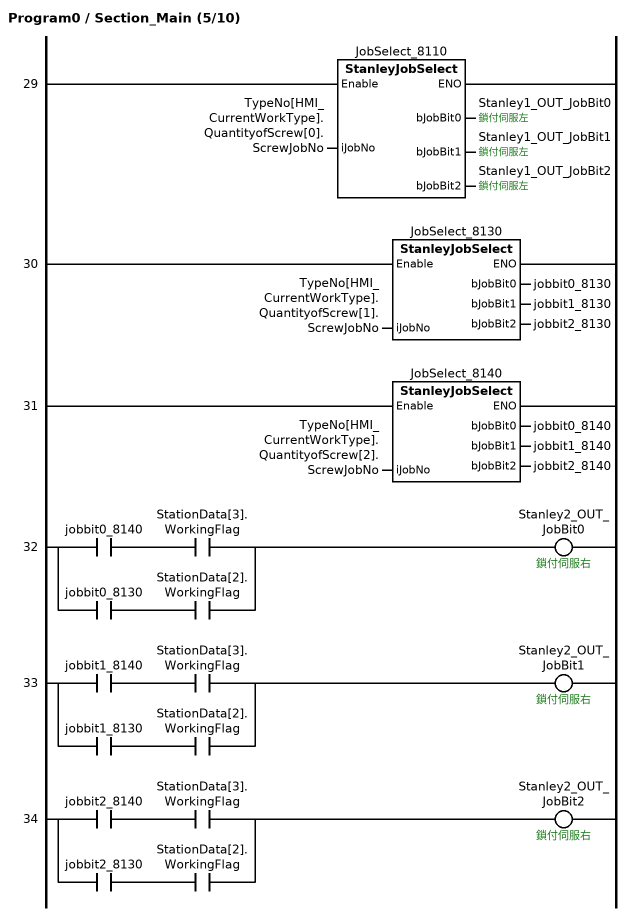
(* Rung 29 *)
JobSelect_8110(Enable := TRUE, iJobNo := TypeNo[HMI_CurrentWorkType].QuantityofScrew[0].ScrewJobNo, bJobBit0 => Stanley1_OUT_JobBit0, bJobBit1 => Stanley1_OUT_JobBit1, bJobBit2 => Stanley1_OUT_JobBit2);
(* Rung 30 *)
JobSelect_8130(Enable := TRUE, iJobNo := TypeNo[HMI_CurrentWorkType].QuantityofScrew[1].ScrewJobNo, bJobBit0 => jobbit0_8130, bJobBit1 => jobbit1_8130, bJobBit2 => jobbit2_8130);
(* Rung 31 *)
JobSelect_8140(Enable := TRUE, iJobNo := TypeNo[HMI_CurrentWorkType].QuantityofScrew[2].ScrewJobNo, bJobBit0 => jobbit0_8140, bJobBit1 => jobbit1_8140, bJobBit2 => jobbit2_8140);
(* Rung 32 *)
Stanley2_OUT_JobBit0 := (jobbit0_8140 AND StationData[3].WorkingFlag) OR (jobbit0_8130 AND StationData[2].WorkingFlag);
(* Rung 33 *)
Stanley2_OUT_JobBit1 := (jobbit1_8140 AND StationData[3].WorkingFlag) OR (jobbit1_8130 AND StationData[2].WorkingFlag);
(* Rung 34 *)
Stanley2_OUT_JobBit2 := (jobbit2_8140 AND StationData[3].WorkingFlag) OR (jobbit2_8130 AND StationData[2].WorkingFlag);

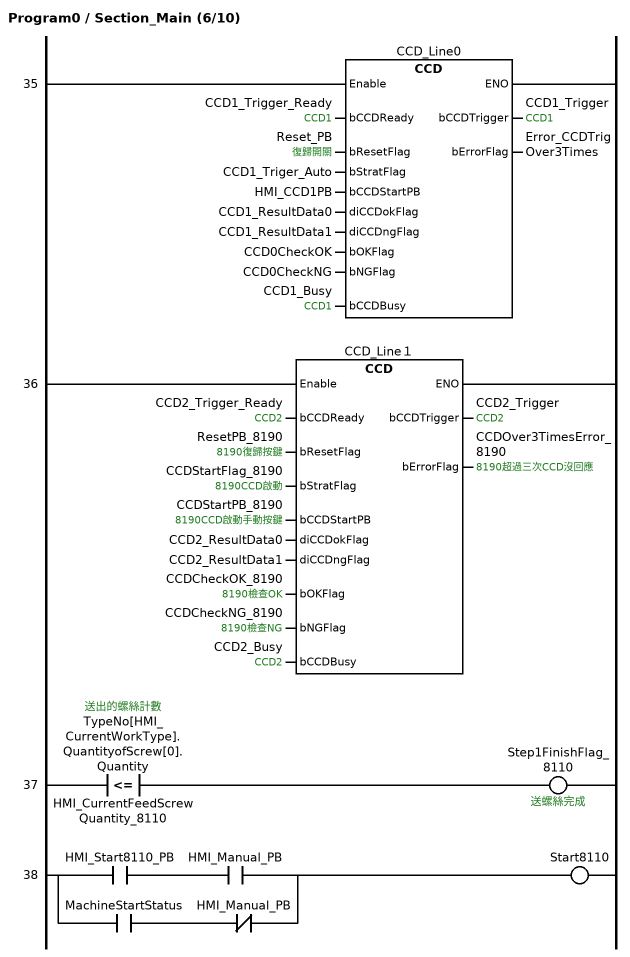
(* Rung 35 *)
CCD_Line0(Enable := TRUE, bCCDReady := CCD1_Trigger_Ready, bResetFlag := Reset_PB, bStratFlag := CCD1_Triger_Auto, bCCDStartPB := HMI_CCD1PB, diCCDokFlag := CCD1_ResultData0, diCCDngFlag := CCD1_ResultData1, bOKFlag := CCD0CheckOK, bNGFlag := CCD0CheckNG, bCCDBusy := CCD1_Busy, bCCDTrigger => CCD1_Trigger, bErrorFlag => Error_CCDTrigOver3Times);
(* Rung 36 *)
CCD_Line１(Enable := TRUE, bCCDReady := CCD2_Trigger_Ready, bResetFlag := ResetPB_8190, bStratFlag := CCDStartFlag_8190, bCCDStartPB := CCDStartPB_8190, diCCDokFlag := CCD2_ResultData0, diCCDngFlag := CCD2_ResultData1, bOKFlag := CCDCheckOK_8190, bNGFlag := CCDCheckNG_8190, bCCDBusy := CCD2_Busy, bCCDTrigger => CCD2_Trigger, bErrorFlag => CCDOver3TimesError_8190);
(* Rung 37 *)
Step1FinishFlag_8110 := TypeNo[HMI_CurrentWorkType].QuantityofScrew[0].Quantity <= HMI_CurrentFeedScrewQuantity_8110;
(* Rung 38 *)
Start8110 := (HMI_Start8110_PB AND HMI_Manual_PB) OR (MachineStartStatus AND NOT HMI_Manual_PB);

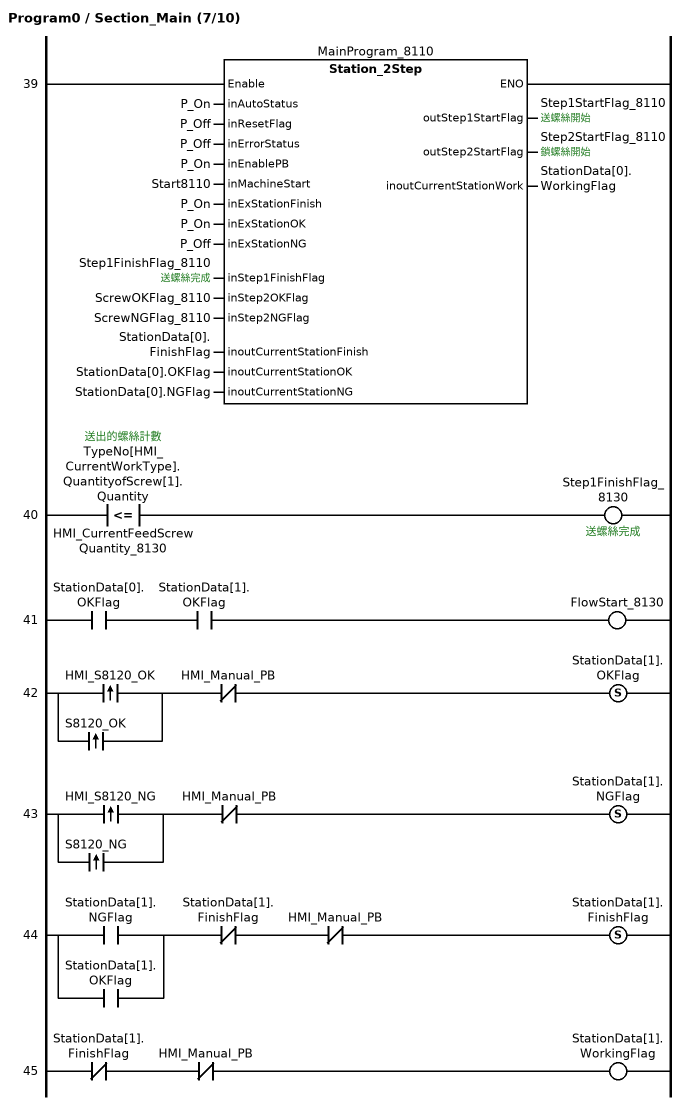
(* Rung 39 *)
MainProgram_8110(Enable := TRUE, inAutoStatus := P_On, inResetFlag := P_Off, inErrorStatus := P_Off, inEnablePB := P_On, inMachineStart := Start8110, inExStationFinish := P_On, inExStationOK := P_On, inExStationNG := P_Off, inStep1FinishFlag := Step1FinishFlag_8110, inStep2OKFlag := ScrewOKFlag_8110, inStep2NGFlag := ScrewNGFlag_8110, inoutCurrentStationFinish := StationData[0].FinishFlag, inoutCurrentStationOK := StationData[0].OKFlag, inoutCurrentStationNG := StationData[0].NGFlag, outStep1StartFlag => Step1StartFlag_8110, outStep2StartFlag => Step2StartFlag_8110, inoutCurrentStationWork => StationData[0].WorkingFlag);
(* Rung 40 *)
Step1FinishFlag_8130 := TypeNo[HMI_CurrentWorkType].QuantityofScrew[1].Quantity <= HMI_CurrentFeedScrewQuantity_8130;
(* Rung 41 *)
FlowStart_8130 := StationData[0].OKFlag AND StationData[1].OKFlag;
(* Rung 42 *)
_e2(CLK := HMI_S8120_OK);
_e3(CLK := S8120_OK);
IF (_e2.Q OR _e3.Q) AND NOT HMI_Manual_PB THEN StationData[1].OKFlag := TRUE; END_IF;
(* Rung 43 *)
_e4(CLK := HMI_S8120_NG);
_e5(CLK := S8120_NG);
IF (_e4.Q OR _e5.Q) AND NOT HMI_Manual_PB THEN StationData[1].NGFlag := TRUE; END_IF;
(* Rung 44 *)
IF (StationData[1].NGFlag OR StationData[1].OKFlag) AND NOT StationData[1].FinishFlag AND NOT HMI_Manual_PB THEN
    StationData[1].FinishFlag := TRUE;
END_IF;
(* Rung 45 *)
StationData[1].WorkingFlag := NOT StationData[1].FinishFlag AND NOT HMI_Manual_PB;

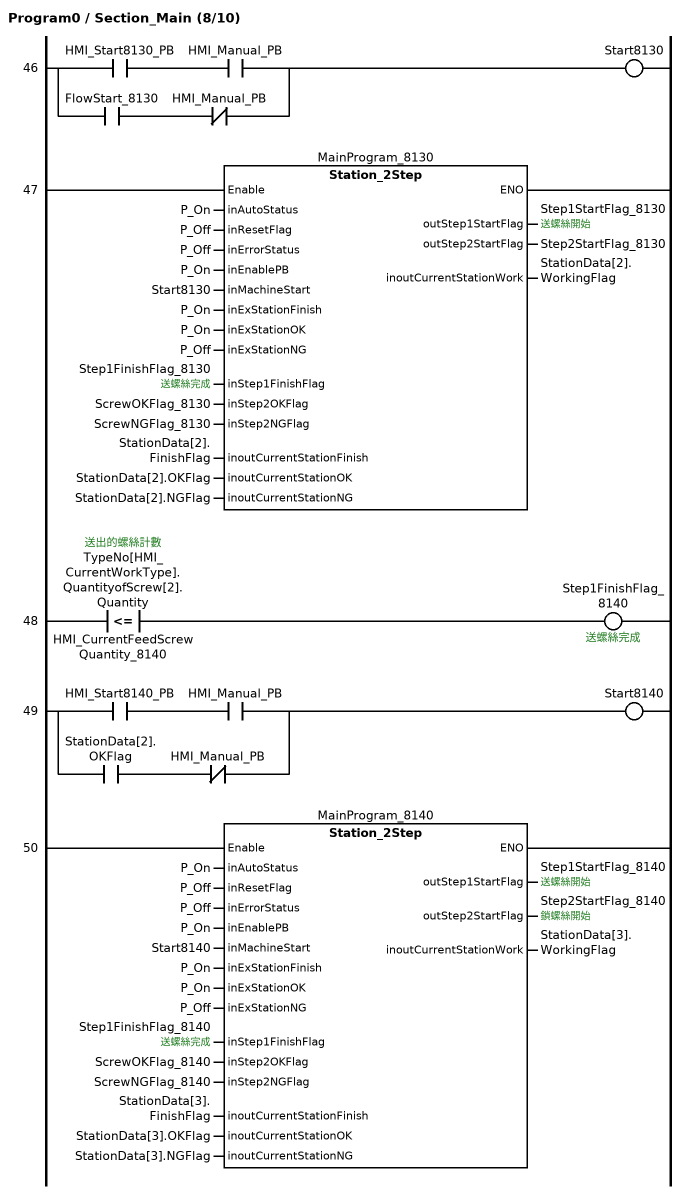
(* Rung 46 *)
Start8130 := (HMI_Start8130_PB AND HMI_Manual_PB) OR (FlowStart_8130 AND NOT HMI_Manual_PB);
(* Rung 47 *)
MainProgram_8130(Enable := TRUE, inAutoStatus := P_On, inResetFlag := P_Off, inErrorStatus := P_Off, inEnablePB := P_On, inMachineStart := Start8130, inExStationFinish := P_On, inExStationOK := P_On, inExStationNG := P_Off, inStep1FinishFlag := Step1FinishFlag_8130, inStep2OKFlag := ScrewOKFlag_8130, inStep2NGFlag := ScrewNGFlag_8130, inoutCurrentStationFinish := StationData[2].FinishFlag, inoutCurrentStationOK := StationData[2].OKFlag, inoutCurrentStationNG := StationData[2].NGFlag, outStep1StartFlag => Step1StartFlag_8130, outStep2StartFlag => Step2StartFlag_8130, inoutCurrentStationWork => StationData[2].WorkingFlag);
(* Rung 48 *)
Step1FinishFlag_8140 := TypeNo[HMI_CurrentWorkType].QuantityofScrew[2].Quantity <= HMI_CurrentFeedScrewQuantity_8140;
(* Rung 49 *)
Start8140 := (HMI_Start8140_PB AND HMI_Manual_PB) OR (StationData[2].OKFlag AND NOT HMI_Manual_PB);
(* Rung 50 *)
MainProgram_8140(Enable := TRUE, inAutoStatus := P_On, inResetFlag := P_Off, inErrorStatus := P_Off, inEnablePB := P_On, inMachineStart := Start8140, inExStationFinish := P_On, inExStationOK := P_On, inExStationNG := P_Off, inStep1FinishFlag := Step1FinishFlag_8140, inStep2OKFlag := ScrewOKFlag_8140, inStep2NGFlag := ScrewNGFlag_8140, inoutCurrentStationFinish := StationData[3].FinishFlag, inoutCurrentStationOK := StationData[3].OKFlag, inoutCurrentStationNG := StationData[3].NGFlag, outStep1StartFlag => Step1StartFlag_8140, outStep2StartFlag => Step2StartFlag_8140, inoutCurrentStationWork => StationData[3].WorkingFlag);

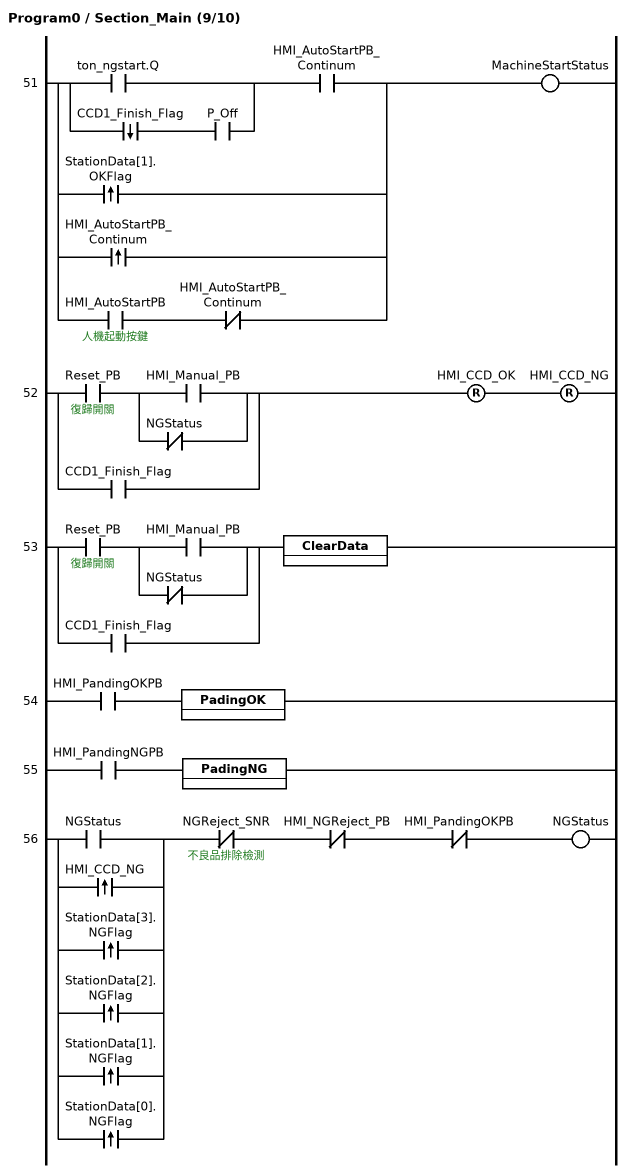
(* Rung 51 *)
_e6(CLK := CCD1_Finish_Flag);
_e7(CLK := StationData[1].OKFlag);
_e8(CLK := HMI_AutoStartPB_Continum);
MachineStartStatus := ((ton_ngstart.Q OR (_e6.Q AND P_Off)) AND HMI_AutoStartPB_Continum) OR _e7.Q OR _e8.Q OR (HMI_AutoStartPB AND NOT HMI_AutoStartPB_Continum);
(* Rung 52 *)
IF (Reset_PB AND (HMI_Manual_PB OR NOT NGStatus)) OR CCD1_Finish_Flag THEN
    HMI_CCD_OK := FALSE;
    HMI_CCD_NG := FALSE;
END_IF;
(* Rung 53 *)
(* drawn but driving nothing: CCD1_Finish_Flag, Reset_PB, NGStatus, HMI_Manual_PB *)
(* Rung 54 *)
(* drawn but driving nothing: HMI_PandingOKPB *)
(* Rung 55 *)
(* drawn but driving nothing: HMI_PandingNGPB *)
(* Rung 56 *)
_e9(CLK := HMI_CCD_NG);
_e10(CLK := StationData[3].NGFlag);
_e11(CLK := StationData[2].NGFlag);
_e12(CLK := StationData[1].NGFlag);
_e13(CLK := StationData[0].NGFlag);
NGStatus := (NGStatus OR _e9.Q OR _e10.Q OR _e11.Q OR _e12.Q OR _e13.Q) AND NOT NGReject_SNR AND NOT HMI_NGReject_PB AND NOT HMI_PandingOKPB;

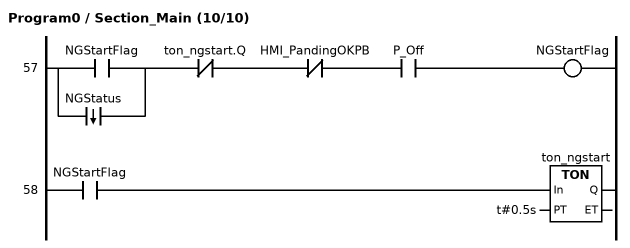
(* Rung 57 *)
_e14(CLK := NGStatus);
NGStartFlag := (NGStartFlag OR _e14.Q) AND NOT ton_ngstart.Q AND NOT HMI_PandingOKPB AND P_Off;
(* Rung 58 *)
ton_ngstart(In := NGStartFlag, PT := t#0.5s);
END_PROGRAM

PROGRAM Program1
VAR
    FeedScrew_1 : FB_FeedScrew_FullBoard;
    FeedScrew_2 : FB_FeedScrew_FullBoard;
    FeedScrew_3 : FB_FeedScrew_FullBoard;
    CheckScrew_1 : FB_CheckScrew;
    CheckScrew_2 : FB_CheckScrew;
    CheckScrew_3 : FB_CheckScrew;
END_VAR
VAR_EXTERNAL
    FeedScrew1_FeedSol : BOOL;
    HMI_FeedScrewPB_1 : BOOL;
    FeedScrew1_FeedRY : BOOL;
    FeedScrew2_FeedSol : BOOL;
    HMI_FeedScrewPB_2 : BOOL;
    FeedScrew2_FeedRY : BOOL;
    FeedScrew3_FeedSol : BOOL;
    HMI_FeedScrewPB_3 : BOOL;
    FeedScrew3_FeedRY : BOOL;
    FeedScrew1_FeedSNR : BOOL;
    Reset_PB : BOOL;
    Error_FeedScrew1_FeedSNR : BOOL;
    FeedScrew2_FeedSNR : BOOL;
    Error_FeedScrew2_FeedSNR : BOOL;
    FeedScrew3_FeedSNR : BOOL;
    Error_FeedScrew3_FeedSNR : BOOL;
    FeedStartFlag_1 : BOOL;
    FeedStartFlag_2 : BOOL;
    FeedStartFlag_3 : BOOL;
END_VAR

(* Section Section_FeedScrew: ladder, written here as Structured Text *)

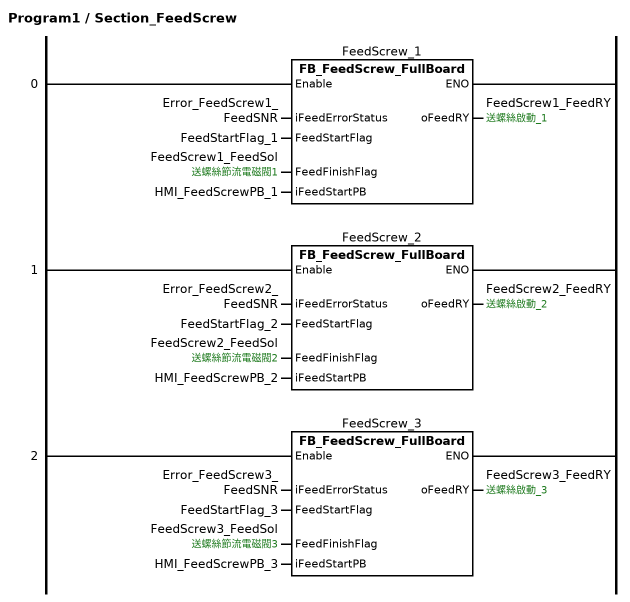
(* Rung 0 *)
FeedScrew_1(Enable := TRUE, iFeedErrorStatus := Error_FeedScrew1_FeedSNR, FeedStartFlag := FeedStartFlag_1, FeedFinishFlag := FeedScrew1_FeedSol, iFeedStartPB := HMI_FeedScrewPB_1, oFeedRY => FeedScrew1_FeedRY);
(* Rung 1 *)
FeedScrew_2(Enable := TRUE, iFeedErrorStatus := Error_FeedScrew2_FeedSNR, FeedStartFlag := FeedStartFlag_2, FeedFinishFlag := FeedScrew2_FeedSol, iFeedStartPB := HMI_FeedScrewPB_2, oFeedRY => FeedScrew2_FeedRY);
(* Rung 2 *)
FeedScrew_3(Enable := TRUE, iFeedErrorStatus := Error_FeedScrew3_FeedSNR, FeedStartFlag := FeedStartFlag_3, FeedFinishFlag := FeedScrew3_FeedSol, iFeedStartPB := HMI_FeedScrewPB_3, oFeedRY => FeedScrew3_FeedRY);

(* Section Section_CheckScrew: ladder, written here as Structured Text *)

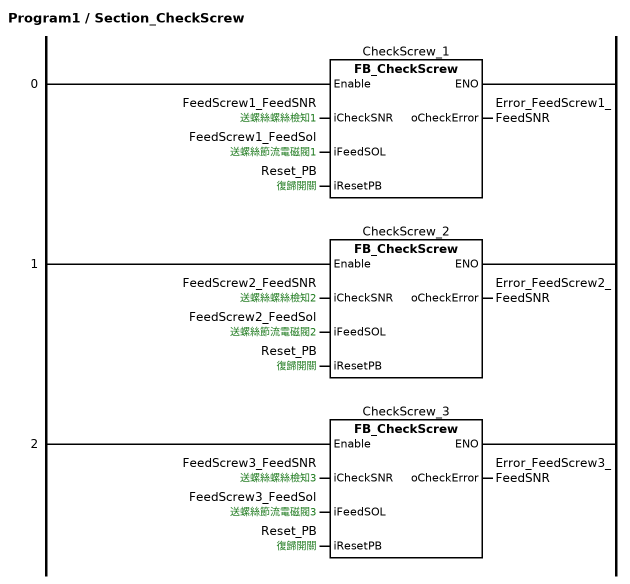
(* Rung 0 *)
CheckScrew_1(Enable := TRUE, iCheckSNR := FeedScrew1_FeedSNR, iFeedSOL := FeedScrew1_FeedSol, iResetPB := Reset_PB, oCheckError => Error_FeedScrew1_FeedSNR);
(* Rung 1 *)
CheckScrew_2(Enable := TRUE, iCheckSNR := FeedScrew2_FeedSNR, iFeedSOL := FeedScrew2_FeedSol, iResetPB := Reset_PB, oCheckError => Error_FeedScrew2_FeedSNR);
(* Rung 2 *)
CheckScrew_3(Enable := TRUE, iCheckSNR := FeedScrew3_FeedSNR, iFeedSOL := FeedScrew3_FeedSol, iResetPB := Reset_PB, oCheckError => Error_FeedScrew3_FeedSNR);
END_PROGRAM

PROGRAM Program2
VAR
    Home_Go : BOOL;
    Zero_Go : BOOL;
    Postion_Go : BOOL;
    Ini : BOOL;
    Ini_state2 : BOOL;
    Ini_state3 : BOOL;
    TON_001 : TON;
    TON_002 : TON;
    TON_003 : TON;
    Ini_state4 : BOOL;
    Jog_CW : BOOL;
    HMI_ASDA_ARSTPB : BOOL;
    ton_1 : TON;
    Init_1 : BOOL;
    ton_p1 : TON;
    Init_2 : BOOL;
    ton_p2 : TON;
    Init_3 : BOOL;
    ton_p3 : TON;
    Init_4 : BOOL;
    ton_p4 : TON;
    Init_5 : BOOL;
    ton_p5 : TON;
    Init_6 : BOOL;
    ton_p6 : TON;
    Init_7 : BOOL;
    ton_p7 : TON;
    Init_8 : BOOL;
    ton_p8 : TON;
    Init_9 : BOOL;
    ton_p9 : TON;
    Init_10 : BOOL;
    ton_p10 : TON;
    MotionSpeed_to_PLC : DINT;
    MotionAddress_to_PLC : DINT;
    timer_PON : TON;
    PowerOn : BOOL;
    Idle : BOOL;
    MotionGoStart_CCD : BOOL;
    MotionGoing_CCD : BOOL;
    MotionGoFinish_CCD : BOOL;
    CCDStart : BOOL;
    CCDing : BOOL;
    CCDFinish : BOOL;
    MotionGoStart_Screw : BOOL;
    MotionGoing_Screw : BOOL;
    MotionGoFinish_Screw : BOOL;
    ton_ServoReady : TON;
    ton_004 : TON;
    MotionGoStart_Reject : BOOL;
    MotionGoing_Reject : BOOL;
    MotionGoFinish_Reject : BOOL;
    Init_11 : BOOL;
    ton_gohome : TON;
END_VAR
VAR_EXTERNAL
    E001_1st_RxPDO_Mapping_Controlword_6040_00 : UINT;
    E001_1st_TxPDO_Mapping_Statusword_6041_00 : UINT;
    Mapping_Controlword_6040_00 : WORD_UNION;
    Mapping_Statusword_6041_00 : WORD_UNION;
    ASDA_OUT_ARST : BOOL;
    E001_1st_RxPDO_Mapping_Modes_of_operation_6060_00 : SINT;
    E001_1st_RxPDO_Mapping_Target_position_607A_00 : DINT;
    E001_1st_RxPDO_Mapping_Profile_velocity_6081_00 : UDINT;
    E001_1st_RxPDO_Mapping_Homing_method_6098_00 : SINT;
    E001_1st_RxPDO_Mapping_Home_offset_607C_00 : DINT;
    HMI_CurrentWorkType : INT;
    TypeNo : ARRAY[0..7] OF WorkType;
    Go_Home : BOOL;
    Go_Zero : BOOL;
    Go_Postion : BOOL;
    ASDA_IN_HOME : BOOL;
    ASDA_IN_ZSPD : BOOL;
    E001_1st_TxPDO_Mapping_Position_actual_value_6064_00 : DINT;
    HMI_CurrentAddress : DINT;
    E001_1st_TxPDO_Mapping_Velocity_actual_value_606C_00 : DINT;
    HMI_CurrentSpeed : DINT;
    Reset_PB : BOOL;
    ASDA_IN_SRDY : BOOL;
    EStop_PB : BOOL;
    StationData : ARRAY[0..3] OF RecordData;
    CCDStart_PB : BOOL;
    CCD1_ResultData0 : DINT;
    HMI_CCD_OK : BOOL;
    HMI_CCD_NG : BOOL;
    CCD1_Trigger_Ready : BOOL;
    E002_Line0_Trigger_Ack : BOOL;
    CCD1_ResultData1 : DINT;
    Go_Zero_Auto : BOOL;
    Go_Position_Auto : BOOL;
    CCD1_Triger_Auto : BOOL;
    CCD1_Finish_Flag : BOOL;
    Go_Home_Auto : BOOL;
    E001_1st_RxPDO_Mapping_Profile_acceleration_6083_00 : UDINT;
    E001_1st_RxPDO_Mapping_Profile_deceleration_6084_00 : UDINT;
    E001_1st_RxPDO_Mapping_Speed_during_search_for_swi_6099_01 : UDINT;
    RejectPosition_Address : DINT;
    Go_Position_Reject : BOOL;
    GoHomedFlag : BOOL;
    S8140OK : BOOL;
    CCDCheckOK_8190 : BOOL;
    CCD0CheckOK : BOOL;
    CCD0CheckNG : BOOL;
    S8140NG : BOOL;
END_VAR
VAR
    _e1 : R_TRIG;
    _e2 : R_TRIG;
    _e3 : R_TRIG;
    _e4 : R_TRIG;
    _e5 : R_TRIG;
    _e6 : R_TRIG;
    _e7 : R_TRIG;
    _e8 : R_TRIG;
    _e9 : F_TRIG;
    _p10 : BOOL;
    _e11 : R_TRIG;
    _e12 : R_TRIG;
    _e13 : R_TRIG;
    _e14 : R_TRIG;
END_VAR

(* Section Section_ServoInit: ladder, written here as Structured Text *)

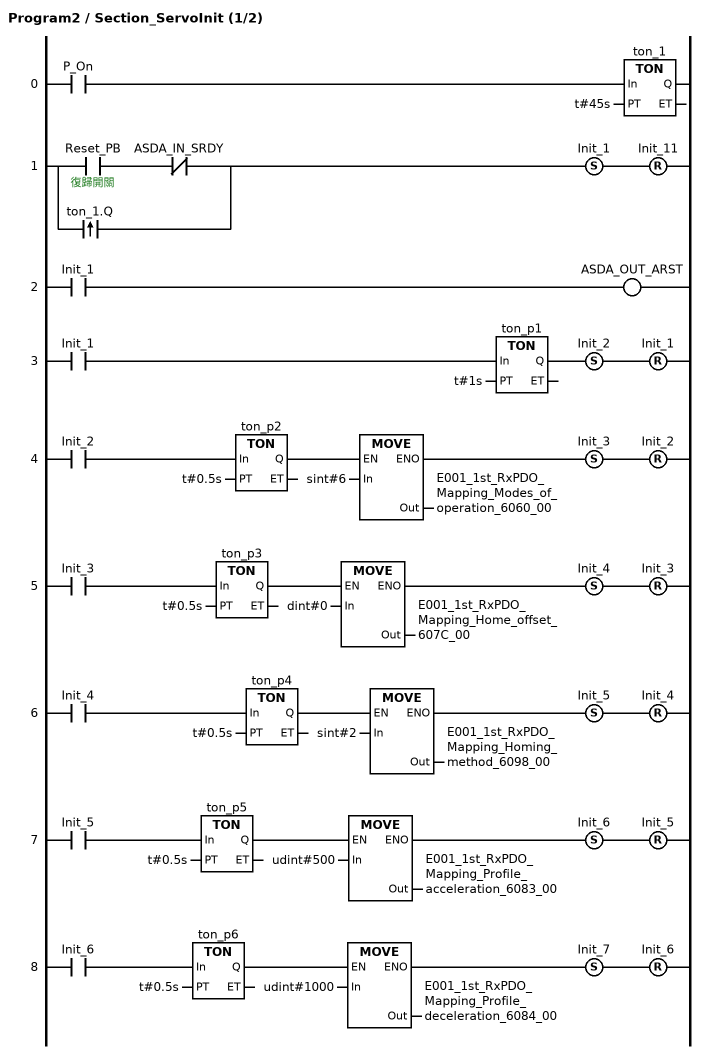
(* Rung 0 *)
ton_1(In := P_On, PT := t#45s);
(* Rung 1 *)
_e1(CLK := ton_1.Q);
IF (Reset_PB AND NOT ASDA_IN_SRDY) OR _e1.Q THEN
    Init_1 := TRUE;
    Init_11 := FALSE;
END_IF;
(* Rung 2 *)
ASDA_OUT_ARST := Init_1;
(* Rung 3 *)
ton_p1(In := Init_1, PT := t#1s);
IF ton_p1.Q THEN
    Init_2 := TRUE;
    Init_1 := FALSE;
END_IF;
(* Rung 4 *)
ton_p2(In := Init_2, PT := t#0.5s);
IF ton_p2.Q THEN
    E001_1st_RxPDO_Mapping_Modes_of_operation_6060_00 := sint#6;
    Init_3 := TRUE;
    Init_2 := FALSE;
END_IF;
(* Rung 5 *)
ton_p3(In := Init_3, PT := t#0.5s);
IF ton_p3.Q THEN
    E001_1st_RxPDO_Mapping_Home_offset_607C_00 := dint#0;
    Init_4 := TRUE;
    Init_3 := FALSE;
END_IF;
(* Rung 6 *)
ton_p4(In := Init_4, PT := t#0.5s);
IF ton_p4.Q THEN
    E001_1st_RxPDO_Mapping_Homing_method_6098_00 := sint#2;
    Init_5 := TRUE;
    Init_4 := FALSE;
END_IF;
(* Rung 7 *)
ton_p5(In := Init_5, PT := t#0.5s);
IF ton_p5.Q THEN
    E001_1st_RxPDO_Mapping_Profile_acceleration_6083_00 := udint#500;
    Init_6 := TRUE;
    Init_5 := FALSE;
END_IF;
(* Rung 8 *)
ton_p6(In := Init_6, PT := t#0.5s);
IF ton_p6.Q THEN
    E001_1st_RxPDO_Mapping_Profile_deceleration_6084_00 := udint#1000;
    Init_7 := TRUE;
    Init_6 := FALSE;
END_IF;

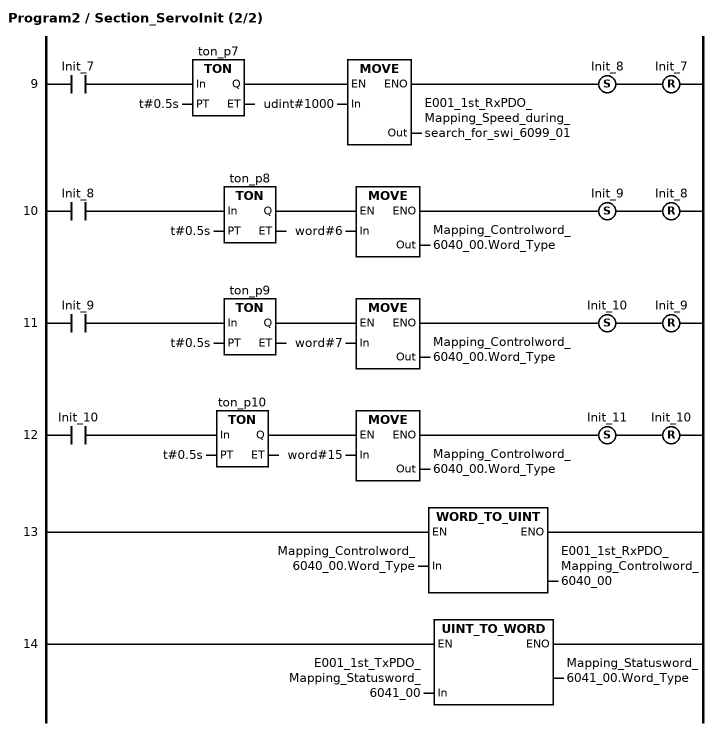
(* Rung 9 *)
ton_p7(In := Init_7, PT := t#0.5s);
IF ton_p7.Q THEN
    E001_1st_RxPDO_Mapping_Speed_during_search_for_swi_6099_01 := udint#1000;
    Init_8 := TRUE;
    Init_7 := FALSE;
END_IF;
(* Rung 10 *)
ton_p8(In := Init_8, PT := t#0.5s);
IF ton_p8.Q THEN
    Mapping_Controlword_6040_00.Word_Type := word#6;
    Init_9 := TRUE;
    Init_8 := FALSE;
END_IF;
(* Rung 11 *)
ton_p9(In := Init_9, PT := t#0.5s);
IF ton_p9.Q THEN
    Mapping_Controlword_6040_00.Word_Type := word#7;
    Init_10 := TRUE;
    Init_9 := FALSE;
END_IF;
(* Rung 12 *)
ton_p10(In := Init_10, PT := t#0.5s);
IF ton_p10.Q THEN
    Mapping_Controlword_6040_00.Word_Type := word#15;
    Init_11 := TRUE;
    Init_10 := FALSE;
END_IF;
(* Rung 13 *)
E001_1st_RxPDO_Mapping_Controlword_6040_00 := WORD_TO_UINT(In := Mapping_Controlword_6040_00.Word_Type);
(* Rung 14 *)
Mapping_Statusword_6041_00.Word_Type := UINT_TO_WORD(In := E001_1st_TxPDO_Mapping_Statusword_6041_00);

(* Section Section_Control: ladder, written here as Structured Text *)

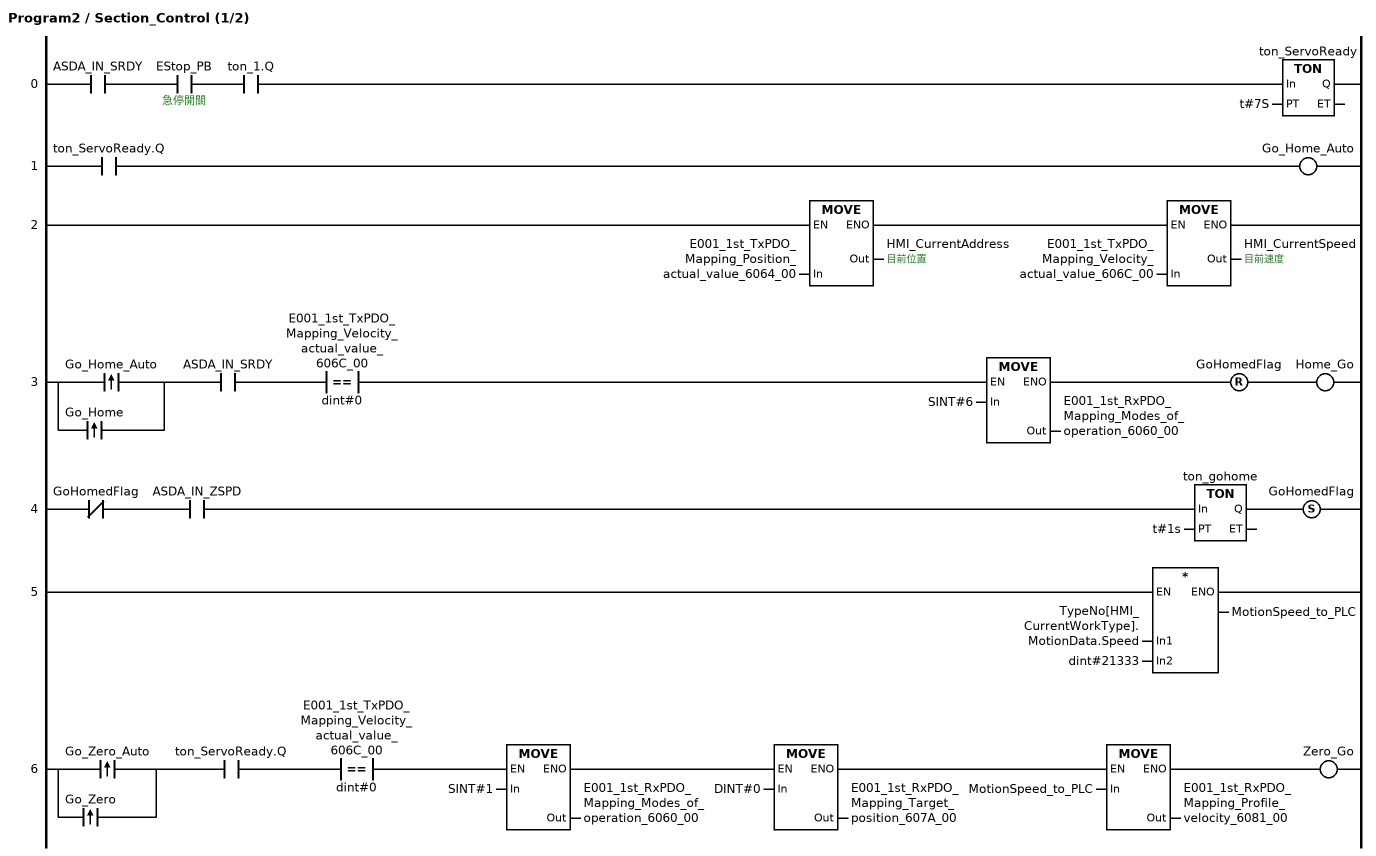
(* Rung 0 *)
ton_ServoReady(In := ASDA_IN_SRDY AND EStop_PB AND ton_1.Q, PT := t#7S);
(* Rung 1 *)
Go_Home_Auto := ton_ServoReady.Q;
(* Rung 2 *)
HMI_CurrentAddress := E001_1st_TxPDO_Mapping_Position_actual_value_6064_00;
HMI_CurrentSpeed := E001_1st_TxPDO_Mapping_Velocity_actual_value_606C_00;
(* Rung 3 *)
_e2(CLK := Go_Home_Auto);
_e3(CLK := Go_Home);
IF (_e2.Q OR _e3.Q) AND ASDA_IN_SRDY AND (E001_1st_TxPDO_Mapping_Velocity_actual_value_606C_00 = dint#0) THEN
    E001_1st_RxPDO_Mapping_Modes_of_operation_6060_00 := SINT#6;
    GoHomedFlag := FALSE;
END_IF;
Home_Go := (_e2.Q OR _e3.Q) AND ASDA_IN_SRDY AND (E001_1st_TxPDO_Mapping_Velocity_actual_value_606C_00 = dint#0);
(* Rung 4 *)
ton_gohome(In := NOT GoHomedFlag AND ASDA_IN_ZSPD, PT := t#1s);
IF ton_gohome.Q THEN GoHomedFlag := TRUE; END_IF;
(* Rung 5 *)
MotionSpeed_to_PLC := TypeNo[HMI_CurrentWorkType].MotionData.Speed * dint#21333;
(* Rung 6 *)
_e4(CLK := Go_Zero_Auto);
_e5(CLK := Go_Zero);
IF (_e4.Q OR _e5.Q) AND ton_ServoReady.Q AND (E001_1st_TxPDO_Mapping_Velocity_actual_value_606C_00 = dint#0) THEN
    E001_1st_RxPDO_Mapping_Modes_of_operation_6060_00 := SINT#1;
    E001_1st_RxPDO_Mapping_Target_position_607A_00 := DINT#0;
    E001_1st_RxPDO_Mapping_Profile_velocity_6081_00 := MotionSpeed_to_PLC;
END_IF;
Zero_Go := (_e4.Q OR _e5.Q) AND ton_ServoReady.Q AND (E001_1st_TxPDO_Mapping_Velocity_actual_value_606C_00 = dint#0);

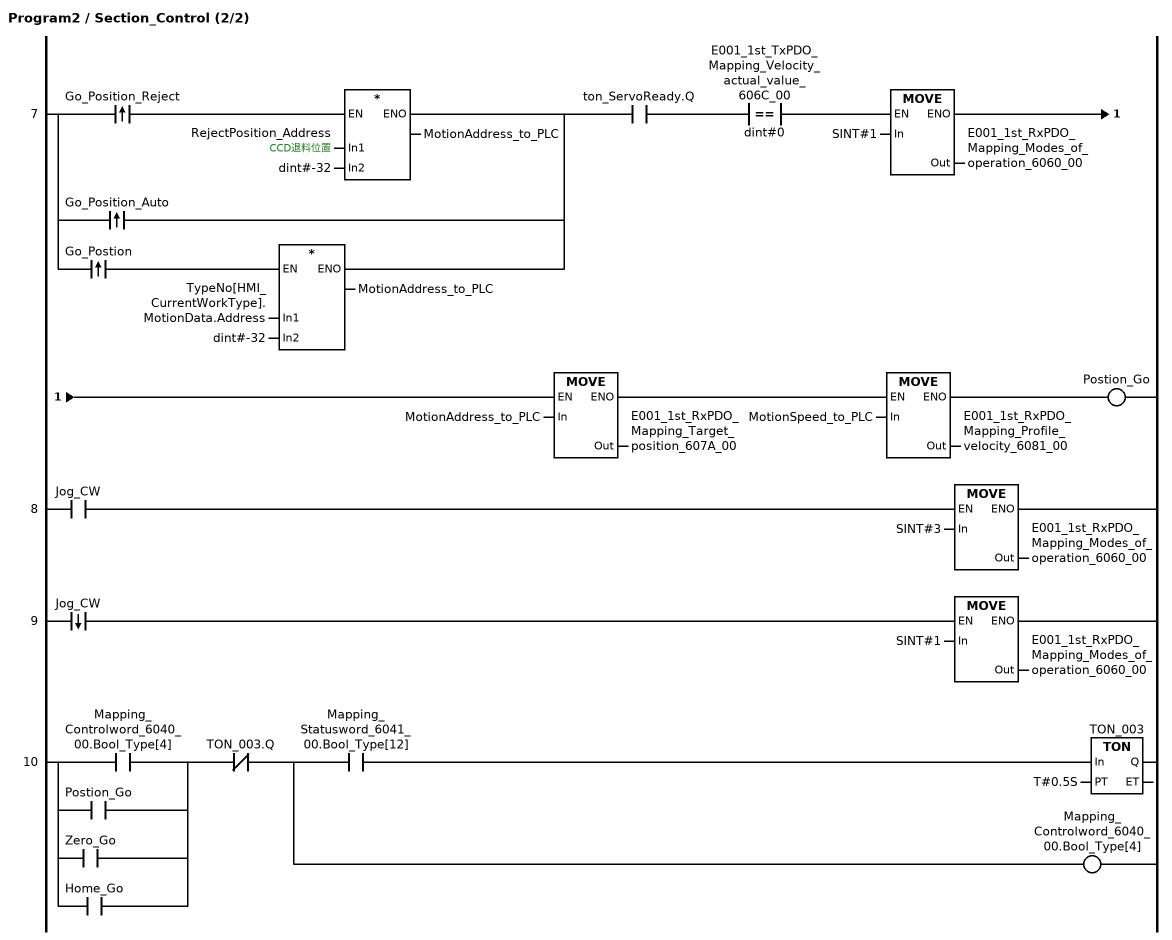
(* Rung 7 *)
_e6(CLK := Go_Position_Reject);
IF _e6.Q THEN MotionAddress_to_PLC := RejectPosition_Address * (dint#-32); END_IF;
_e7(CLK := Go_Position_Auto);
_e8(CLK := Go_Postion);
IF _e8.Q THEN MotionAddress_to_PLC := TypeNo[HMI_CurrentWorkType].MotionData.Address * (dint#-32); END_IF;
IF (_e6.Q OR _e7.Q OR _e8.Q) AND ton_ServoReady.Q AND (E001_1st_TxPDO_Mapping_Velocity_actual_value_606C_00 = dint#0) THEN
    E001_1st_RxPDO_Mapping_Modes_of_operation_6060_00 := SINT#1;
    E001_1st_RxPDO_Mapping_Target_position_607A_00 := MotionAddress_to_PLC;
    E001_1st_RxPDO_Mapping_Profile_velocity_6081_00 := MotionSpeed_to_PLC;
END_IF;
Postion_Go := (_e6.Q OR _e7.Q OR _e8.Q) AND ton_ServoReady.Q AND (E001_1st_TxPDO_Mapping_Velocity_actual_value_606C_00 = dint#0);
(* Rung 8 *)
IF Jog_CW THEN E001_1st_RxPDO_Mapping_Modes_of_operation_6060_00 := SINT#3; END_IF;
(* Rung 9 *)
_e9(CLK := Jog_CW);
IF _e9.Q THEN E001_1st_RxPDO_Mapping_Modes_of_operation_6060_00 := SINT#1; END_IF;
(* Rung 10 *)
_p10 := (Mapping_Controlword_6040_00.Bool_Type[4] OR Postion_Go OR Zero_Go OR Home_Go) AND NOT TON_003.Q;
TON_003(In := _p10 AND Mapping_Statusword_6041_00.Bool_Type[12], PT := T#0.5S);
Mapping_Controlword_6040_00.Bool_Type[4] := _p10;

(* Section Section_CCDMainProgram: ladder, written here as Structured Text *)

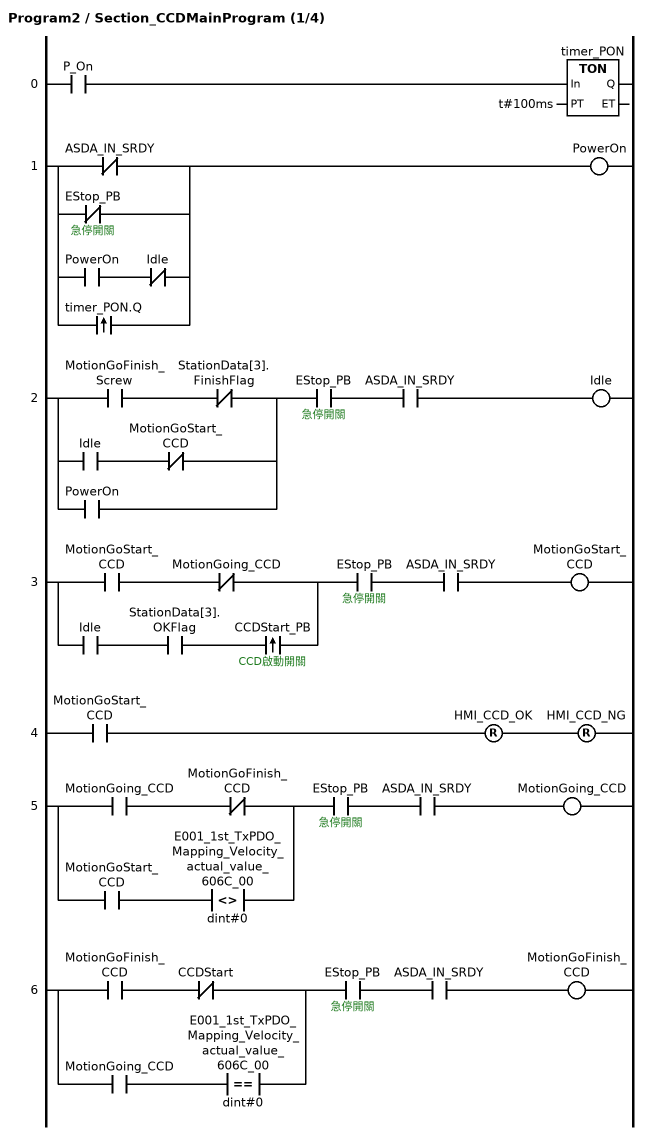
(* Rung 0 *)
timer_PON(In := P_On, PT := t#100ms);
(* Rung 1 *)
_e11(CLK := timer_PON.Q);
PowerOn := NOT ASDA_IN_SRDY OR NOT EStop_PB OR (PowerOn AND NOT Idle) OR _e11.Q;
(* Rung 2 *)
Idle := ((MotionGoFinish_Screw AND NOT StationData[3].FinishFlag) OR (Idle AND NOT MotionGoStart_CCD) OR PowerOn) AND EStop_PB AND ASDA_IN_SRDY;
(* Rung 3 *)
_e12(CLK := CCDStart_PB);
MotionGoStart_CCD := ((MotionGoStart_CCD AND NOT MotionGoing_CCD) OR (Idle AND StationData[3].OKFlag AND _e12.Q)) AND EStop_PB AND ASDA_IN_SRDY;
(* Rung 4 *)
IF MotionGoStart_CCD THEN
    HMI_CCD_OK := FALSE;
    HMI_CCD_NG := FALSE;
END_IF;
(* Rung 5 *)
MotionGoing_CCD := ((MotionGoing_CCD AND NOT MotionGoFinish_CCD) OR (MotionGoStart_CCD AND (E001_1st_TxPDO_Mapping_Velocity_actual_value_606C_00 <> dint#0))) AND EStop_PB AND ASDA_IN_SRDY;
(* Rung 6 *)
MotionGoFinish_CCD := ((MotionGoFinish_CCD AND NOT CCDStart) OR (MotionGoing_CCD AND (E001_1st_TxPDO_Mapping_Velocity_actual_value_606C_00 = dint#0))) AND EStop_PB AND ASDA_IN_SRDY;

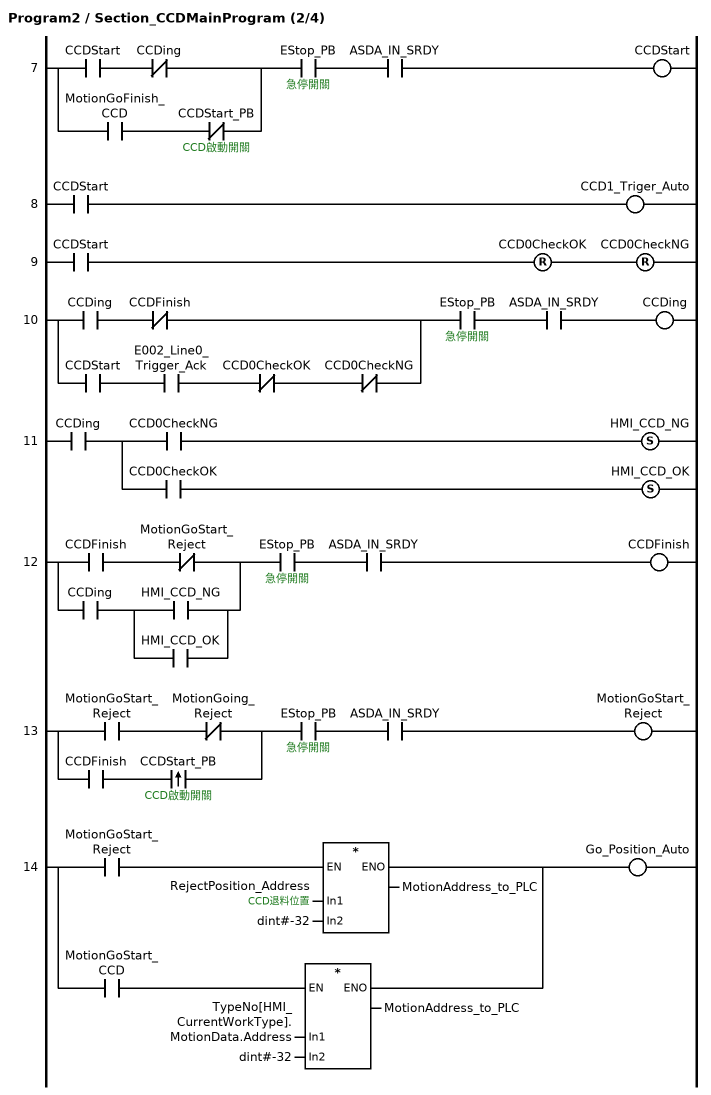
(* Rung 7 *)
CCDStart := ((CCDStart AND NOT CCDing) OR (MotionGoFinish_CCD AND NOT CCDStart_PB)) AND EStop_PB AND ASDA_IN_SRDY;
(* Rung 8 *)
CCD1_Triger_Auto := CCDStart;
(* Rung 9 *)
IF CCDStart THEN
    CCD0CheckOK := FALSE;
    CCD0CheckNG := FALSE;
END_IF;
(* Rung 10 *)
CCDing := ((CCDing AND NOT CCDFinish) OR (CCDStart AND E002_Line0_Trigger_Ack AND NOT CCD0CheckOK AND NOT CCD0CheckNG)) AND EStop_PB AND ASDA_IN_SRDY;
(* Rung 11 *)
IF CCDing AND CCD0CheckNG THEN HMI_CCD_NG := TRUE; END_IF;
IF CCDing AND CCD0CheckOK THEN HMI_CCD_OK := TRUE; END_IF;
(* Rung 12 *)
CCDFinish := ((CCDFinish AND NOT MotionGoStart_Reject) OR (CCDing AND (HMI_CCD_NG OR HMI_CCD_OK))) AND EStop_PB AND ASDA_IN_SRDY;
(* Rung 13 *)
_e13(CLK := CCDStart_PB);
MotionGoStart_Reject := ((MotionGoStart_Reject AND NOT MotionGoing_Reject) OR (CCDFinish AND _e13.Q)) AND EStop_PB AND ASDA_IN_SRDY;
(* Rung 14 *)
IF MotionGoStart_Reject THEN MotionAddress_to_PLC := RejectPosition_Address * (dint#-32); END_IF;
IF MotionGoStart_CCD THEN
    MotionAddress_to_PLC := TypeNo[HMI_CurrentWorkType].MotionData.Address * (dint#-32);
END_IF;
Go_Position_Auto := MotionGoStart_Reject OR MotionGoStart_CCD;

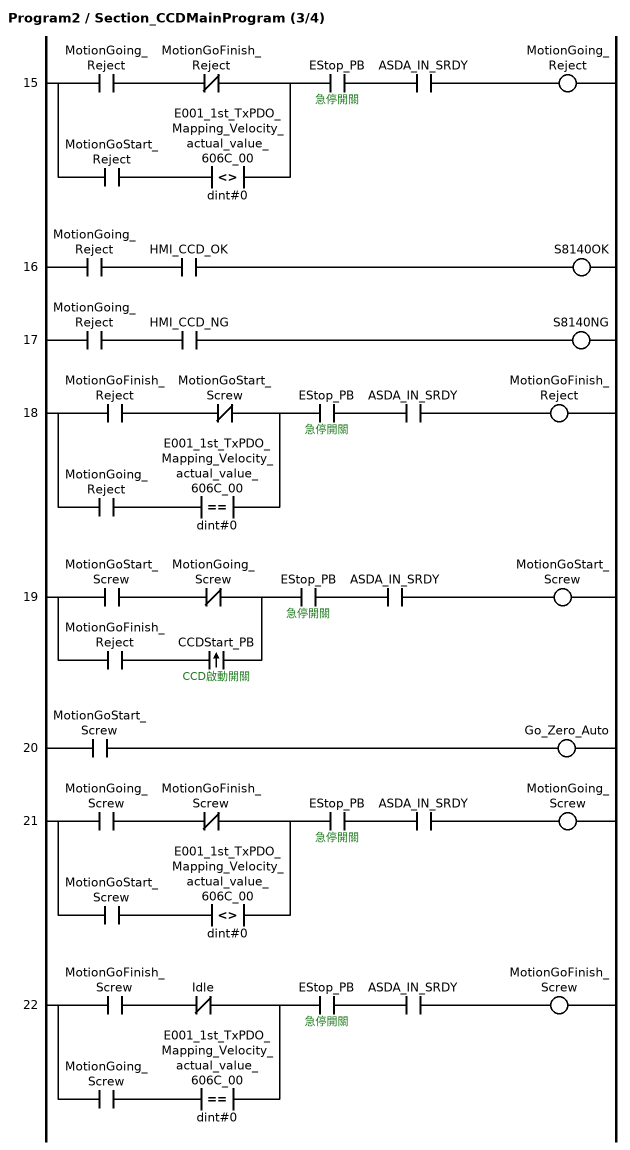
(* Rung 15 *)
MotionGoing_Reject := ((MotionGoing_Reject AND NOT MotionGoFinish_Reject) OR (MotionGoStart_Reject AND (E001_1st_TxPDO_Mapping_Velocity_actual_value_606C_00 <> dint#0))) AND EStop_PB AND ASDA_IN_SRDY;
(* Rung 16 *)
S8140OK := MotionGoing_Reject AND HMI_CCD_OK;
(* Rung 17 *)
S8140NG := MotionGoing_Reject AND HMI_CCD_NG;
(* Rung 18 *)
MotionGoFinish_Reject := ((MotionGoFinish_Reject AND NOT MotionGoStart_Screw) OR (MotionGoing_Reject AND (E001_1st_TxPDO_Mapping_Velocity_actual_value_606C_00 = dint#0))) AND EStop_PB AND ASDA_IN_SRDY;
(* Rung 19 *)
_e14(CLK := CCDStart_PB);
MotionGoStart_Screw := ((MotionGoStart_Screw AND NOT MotionGoing_Screw) OR (MotionGoFinish_Reject AND _e14.Q)) AND EStop_PB AND ASDA_IN_SRDY;
(* Rung 20 *)
Go_Zero_Auto := MotionGoStart_Screw;
(* Rung 21 *)
MotionGoing_Screw := ((MotionGoing_Screw AND NOT MotionGoFinish_Screw) OR (MotionGoStart_Screw AND (E001_1st_TxPDO_Mapping_Velocity_actual_value_606C_00 <> dint#0))) AND EStop_PB AND ASDA_IN_SRDY;
(* Rung 22 *)
MotionGoFinish_Screw := ((MotionGoFinish_Screw AND NOT Idle) OR (MotionGoing_Screw AND (E001_1st_TxPDO_Mapping_Velocity_actual_value_606C_00 = dint#0))) AND EStop_PB AND ASDA_IN_SRDY;

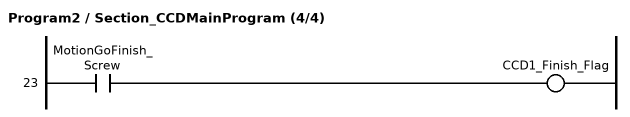
(* Rung 23 *)
CCD1_Finish_Flag := MotionGoFinish_Screw;
END_PROGRAM

PROGRAM prS8120CCD
VAR
    AutoFlow : INT := 0;
    TON_Auto : ARRAY[0..1] OF TON;
    TON_Q : ARRAY[0..1] OF BOOL;
    TON_ET : ARRAY[0..1] OF TIME;
    SectionChangeFlow : INT;
    TON_SectionChange : ARRAY[0..1] OF TON;
    var2 : BOOL;
    var3 : TIME;
    SectionChangeFlow2 : INT;
    var4 : BOOL;
    var5 : TIME;
    OK_Q : BOOL;
    OK_ET : TIME;
    NG_Q : BOOL;
    NG_ET : TIME;
    TON_OK : TON;
    TON_NG : TON;
END_VAR
VAR_EXTERNAL
    HMI_8120CCDBackPB : BOOL;
    HMI_8120CCDOutPB : BOOL;
    Check8120Back_SOL : BOOL;
    Check8120Out_SOL : BOOL;
    Check8120Back_LS : BOOL;
    Check8120Out_LS : BOOL;
    HMI_8120STARTPB : BOOL;
    StationData : ARRAY[0..3] OF RecordData;
    Check8120_CCDTrig : BOOL;
    Check8120_CCDBusy : BOOL;
    Check8120_CCDNG : BOOL;
    S8120_NG : BOOL;
    S8120_OK : BOOL;
    HMI_8120CCDstartPB : BOOL;
    HMI_S8120_OK : BOOL;
    HMI_S8120_NG : BOOL;
    Check8120_CCDStartPB : BOOL;
    E002_Line0_Command_Ready : BOOL;
    CCDSectionChangeFlag : BOOL;
    E002_Line0_Command_Parameter_0 : DINT;
    TypeNo : ARRAY[0..7] OF WorkType;
    E002_Line0_Command_Code : DWORD;
    E002_Line0_Command_Request : BOOL;
    E002_Line0_Command_Completion : BOOL;
    HMI_CurrentWorkType : INT;
    E002_Line1_Command_Ready : BOOL;
    CCDSectionChange : BOOL;
    E002_Line1_Command_Parameter_0 : DINT;
    CCDSectionNo : INT;
    E002_Line1_Command_Code : DWORD;
    E002_Line1_Command_Request : BOOL;
    E002_Line1_Command_Completion : BOOL;
    CCDSectionChangeComplete : BOOL;
    FQ2_Busy : BOOL;
    FQ2_NG : BOOL;
END_VAR
//HMI訊號
FQ2_Busy:=Check8120_CCDBusy;
FQ2_NG:=Check8120_CCDNG;
(***************************************************************)
//程序名稱:8120加CCD
//作者:蔡相偉
//日期:2016/5/4  版本:v1.0
//PowerOn=0
//Idle=1
//移位出=2
//CCD開始=3
//CCD拍攝中=4
//CCD完成=5
//移位回=6
(***************************************************************)
//PowerOn=0
TON_Auto[0](In:=AutoFlow=0, PT:=t#10ms, Q=>TON_Q[0], ET=>TON_ET[0]);

IF AutoFlow=0 AND TON_Q[0] THEN
	AutoFlow:=1;	
END_IF;
//Idle=1

IF AutoFlow=1 AND Check8120_CCDStartPB THEN
	AutoFlow:=2;
END_IF;
//移位出=2
IF AutoFlow=2 THEN
	HMI_S8120_NG:=FALSE;
	HMI_S8120_OK:=FALSE;
	StationData[1].OKFlag:=FALSE;
	StationData[1].NGFlag:=FALSE;
	StationData[1].FinishFlag:=FALSE;
END_IF;

IF AutoFlow=2 AND Check8120Out_LS AND NOT(HMI_S8120_NG) AND NOT(HMI_S8120_OK) THEN
	AutoFlow:=3;
END_IF;
//CCD開始=3
IF AutoFlow=3 AND Check8120_CCDBusy THEN
	AutoFlow:=4;
END_IF;
//CCD拍攝中=4
IF AutoFlow=4 AND NOT(Check8120_CCDBusy) THEN
	AutoFlow:=5;
END_IF;
//CCD完成=5
TON_OK(In:=AutoFlow=5 AND not(Check8120_CCDNG), PT:=T#30ms, Q=>OK_Q, ET=>OK_ET);
TON_NG(In:=AutoFlow=5 AND Check8120_CCDNG, PT:=T#30ms, Q=>NG_Q, ET=>NG_ET);
IF AutoFlow=5 THEN
	IF NG_Q THEN
		HMI_S8120_NG:=TRUE;
		HMI_S8120_OK:=FALSE;
	END_IF;
	IF OK_Q THEN
		HMI_S8120_NG:=FALSE;
		HMI_S8120_OK:=TRUE;
	END_IF;
END_IF;

IF AutoFlow=5 AND (HMI_S8120_NG OR HMI_S8120_OK) THEN
	AutoFlow:=6;
END_IF;
//移位回=6
IF AutoFlow=6 AND Check8120Back_LS THEN
	//HMI_S8120_NG:=FALSE;
	//HMI_S8120_OK:=FALSE;
	AutoFlow:=1;
END_IF;
(*************************手動*********************************)
//移位歸
//SET
if HMI_8120CCDBackPB OR AutoFlow=6 THEN
	Check8120Back_SOL:=TRUE;
	Check8120Out_SOL:=FALSE;
END_IF;
//RESET
IF Check8120Back_LS THEN
	Check8120Back_SOL:=FALSE;
END_IF;
//移位出
//SET
if HMI_8120CCDOutPB OR AutoFlow=2 THEN
	Check8120Back_SOL:=FALSE;
	Check8120Out_SOL:=TRUE;
END_IF;
//RESET
IF Check8120Out_LS THEN
	Check8120Out_SOL:=FALSE;
END_IF;
//CCD
IF HMI_8120CCDstartPB OR AutoFlow=3 THEN
	Check8120_CCDTrig:=TRUE;
ELSE
	Check8120_CCDTrig:=FALSE;
END_IF;
(*************************手動*********************************)
(***************************************************************)
//程序名稱:場景切換CCD0
//作者:蔡相偉
//日期:2016/5/5  版本:v1.0
//PowerOn=0
//Idle=1
//復制場景編號=2
//復制命令=3
//命令請求=4
//命令完成=5
(***************************************************************)
//PowerOn=0
TON_SectionChange[0](In:=SectionChangeFlow=0, PT:=t#1s, Q=>var2, ET=>var3);
IF var2 THEN
	SectionChangeFlow:=1;
END_IF;
//Idle=1
IF SectionChangeFlow=1 AND E002_Line0_Command_Ready AND CCDSectionChangeFlag  THEN
	SectionChangeFlow:=2;
END_IF;
//復制場景編號=2
IF SectionChangeFlow=2 THEN
	E002_Line0_Command_Parameter_0:=INT_TO_DINT(TypeNo[HMI_CurrentWorkType].CCDSectionNo);
END_IF;

IF SectionChangeFlow=2 AND (E002_Line0_Command_Parameter_0=TypeNo[HMI_CurrentWorkType].CCDSectionNo) THEN
	SectionChangeFlow:=3;
END_IF;
//復制命令=3
IF SectionChangeFlow=3 THEN
	E002_Line0_Command_Code:=16#00301000;
END_IF;
IF SectionChangeFlow=3 AND (E002_Line0_Command_Code=16#00301000) THEN
	SectionChangeFlow:=4;
END_IF;
//命令請求=4
IF SectionChangeFlow=4 THEN
	E002_Line0_Command_Request:=TRUE;
ELSE
	E002_Line0_Command_Request:=FALSE;
END_IF;

IF SectionChangeFlow=4 AND E002_Line0_Command_Completion THEN
	SectionChangeFlow:=5;
END_IF;
//命令完成=5
IF SectionChangeFlow=5 AND NOT(E002_Line0_Command_Completion) THEN
	CCDSectionChangeFlag:=FALSE;
	SectionChangeFlow:=1;
END_IF;

(***************************************************************)
(***************************************************************)
//程序名稱:場景切換CCD1
//作者:蔡相偉
//日期:2016/5/5  版本:v1.0
//PowerOn=0
//Idle=1
//復制場景編號=2
//復制命令=3
//命令請求=4
//命令完成=5
(***************************************************************)
//PowerOn=0
TON_SectionChange[1](In:=SectionChangeFlow2=0, PT:=t#1s, Q=>var4, ET=>var5);
IF var4 THEN
	SectionChangeFlow2:=1;
END_IF;
//Idle=1
IF SectionChangeFlow2=1 AND E002_Line1_Command_Ready AND CCDSectionChange  THEN
	SectionChangeFlow2:=2;
END_IF;
//復制場景編號=2
IF SectionChangeFlow2=2 THEN
	E002_Line1_Command_Parameter_0:=INT_TO_DINT(CCDSectionNo);
END_IF;

IF SectionChangeFlow2=2 AND (E002_Line1_Command_Parameter_0=CCDSectionNo) THEN
	SectionChangeFlow2:=3;
END_IF;
//復制命令=3
IF SectionChangeFlow2=3 THEN
	E002_Line1_Command_Code:=16#00301000;
END_IF;
IF SectionChangeFlow2=3 AND (E002_Line1_Command_Code=16#00301000) THEN
	SectionChangeFlow2:=4;
END_IF;
//命令請求=4
IF SectionChangeFlow2=4 THEN
	E002_Line1_Command_Request:=TRUE;
ELSE
	E002_Line1_Command_Request:=FALSE;
END_IF;

IF SectionChangeFlow2=4 AND E002_Line1_Command_Completion THEN
	SectionChangeFlow2:=5;
END_IF;
//命令完成=5
IF SectionChangeFlow2=5 THEN
	CCDSectionChangeComplete:=TRUE;
ELSE
	CCDSectionChangeComplete:=FALSE;
END_IF;
IF SectionChangeFlow2=5 AND NOT(E002_Line1_Command_Completion) AND NOT(CCDSectionChange) THEN
	SectionChangeFlow2:=1;
END_IF;

(***************************************************************)
END_PROGRAM

FUNCTION ClearData : BOOL
VAR
    ii : INT;
END_VAR
VAR_EXTERNAL
    StationData : ARRAY[0..3] OF RecordData;
END_VAR
FOR ii:=0 TO 3 BY 1 DO
    StationData[ii].NGFlag:=FALSE;
	StationData[ii].OKFlag:=FALSE;
	StationData[ii].FinishFlag:=FALSE;	
END_FOR;
END_FUNCTION

FUNCTION PadingOK : BOOL
VAR_EXTERNAL
    StationData : ARRAY[0..3] OF RecordData;
END_VAR
IF StationData[3].NGFlag THEN
    StationData[3].NGFlag:=FALSE;
	StationData[3].OKFlag:=TRUE;
END_IF;
IF StationData[2].NGFlag THEN
    StationData[2].NGFlag:=FALSE;
	StationData[2].OKFlag:=TRUE;
END_IF;
IF StationData[1].NGFlag THEN
    StationData[1].NGFlag:=FALSE;
	StationData[1].OKFlag:=TRUE;
END_IF;
IF StationData[0].NGFlag THEN
	StationData[0].NGFlag:=FALSE;
	StationData[0].OKFlag:=TRUE;
END_IF;
END_FUNCTION

FUNCTION PadingNG : BOOL
VAR_EXTERNAL
    StationData : ARRAY[0..3] OF RecordData;
END_VAR
IF StationData[3].OKFlag THEN
    StationData[3].NGFlag:=TRUE;
	StationData[3].OKFlag:=FALSE;
END_IF;
IF StationData[2].OKFlag THEN
    StationData[2].NGFlag:=TRUE;
	StationData[2].OKFlag:=FALSE;
END_IF;
IF StationData[1].OKFlag THEN
    StationData[1].NGFlag:=TRUE;
	StationData[1].OKFlag:=FALSE;
END_IF;
IF StationData[0].OKFlag THEN
	StationData[0].NGFlag:=TRUE;
	StationData[0].OKFlag:=FALSE;
END_IF;
END_FUNCTION

FUNCTION_BLOCK FB_FeedScrew_FullBoard
(* 此FB用在單軸電路板,利用繼電器AB接點切換,做送螺絲動作 *)
VAR
    PowerOn : BOOL;
    Idle : BOOL;
    TON_PowerOn : TON;
    FeedStart : BOOL;
    FeedFinish : BOOL;
    RelayOn : BOOL;
    TON_FeedStart : TON;
    RelayOff : BOOL;
    TON_RelayOn : TON;
    TON_RelayOff : TON;
    TON_PON : TON;
END_VAR
VAR_INPUT
    Enable : BOOL;
    iFeedErrorStatus : BOOL;
    FeedStartFlag : BOOL;  (* 送螺絲起動旗標 *)
    FeedFinishFlag : BOOL;  (* 節流電磁閥 *)
    iFeedStartPB : BOOL;  (* 送螺絲手動起動 *)
END_VAR
VAR_OUTPUT
    oFeedRY : BOOL;  (* 繼電器_用在電路板上 *)
END_VAR
VAR
    _e1 : R_TRIG;
END_VAR
(* ladder, written here as Structured Text *)

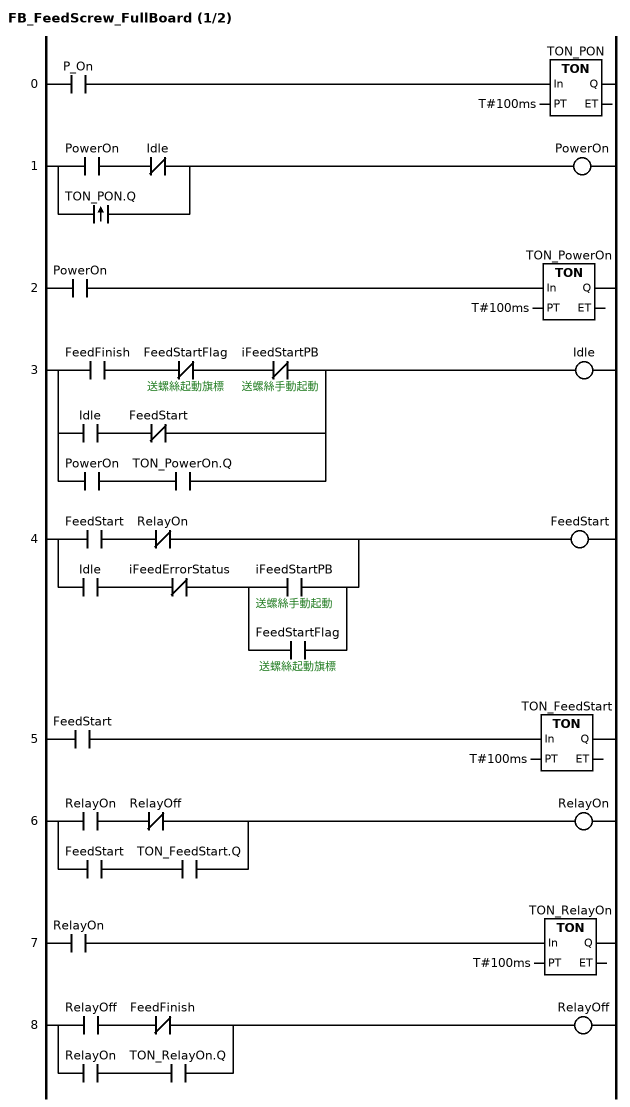
(* Rung 0 *)
TON_PON(In := P_On, PT := T#100ms);
(* Rung 1 *)
_e1(CLK := TON_PON.Q);
PowerOn := (PowerOn AND NOT Idle) OR _e1.Q;
(* Rung 2 *)
TON_PowerOn(In := PowerOn, PT := T#100ms);
(* Rung 3 *)
Idle := (FeedFinish AND NOT FeedStartFlag AND NOT iFeedStartPB) OR (Idle AND NOT FeedStart) OR (PowerOn AND TON_PowerOn.Q);
(* Rung 4 *)
FeedStart := (FeedStart AND NOT RelayOn) OR (Idle AND NOT iFeedErrorStatus AND (iFeedStartPB OR FeedStartFlag));
(* Rung 5 *)
TON_FeedStart(In := FeedStart, PT := T#100ms);
(* Rung 6 *)
RelayOn := (RelayOn AND NOT RelayOff) OR (FeedStart AND TON_FeedStart.Q);
(* Rung 7 *)
TON_RelayOn(In := RelayOn, PT := T#100ms);
(* Rung 8 *)
RelayOff := (RelayOff AND NOT FeedFinish) OR (RelayOn AND TON_RelayOn.Q);

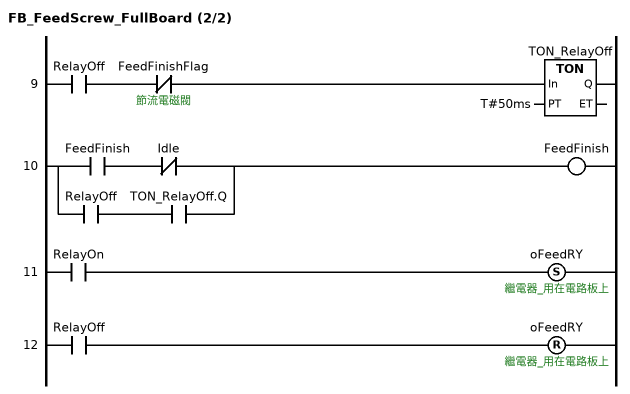
(* Rung 9 *)
TON_RelayOff(In := RelayOff AND NOT FeedFinishFlag, PT := T#50ms);
(* Rung 10 *)
FeedFinish := (FeedFinish AND NOT Idle) OR (RelayOff AND TON_RelayOff.Q);
(* Rung 11 *)
IF RelayOn THEN oFeedRY := TRUE; END_IF;
(* Rung 12 *)
IF RelayOff THEN oFeedRY := FALSE; END_IF;
END_FUNCTION_BLOCK

FUNCTION_BLOCK FB_CheckScrew
(* 檢查螺絲是否送出至夾頭 *)
VAR RETAIN
    ScrewInTube : INT;
    ScrewInClamp : INT;
END_VAR
VAR_INPUT
    Enable : BOOL;
    iCheckSNR : BOOL;  (* 缺螺絲檢知 *)
    iFeedSOL : BOOL;
    iResetPB : BOOL;
END_VAR
VAR_OUTPUT
    oCheckError : BOOL;
END_VAR
VAR
    _e1 : R_TRIG;
    _e2 : R_TRIG;
END_VAR
(* ladder, written here as Structured Text *)

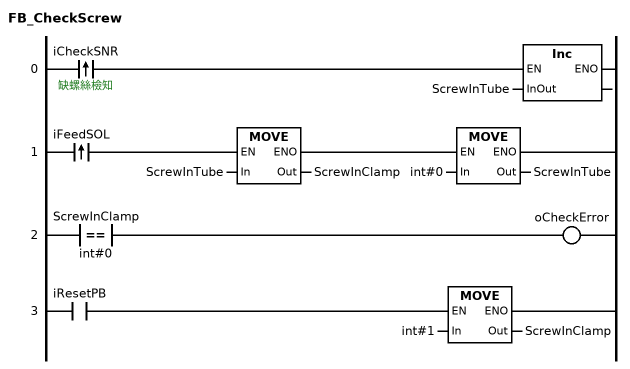
(* Rung 0 *)
_e1(CLK := iCheckSNR);
IF _e1.Q THEN Inc(InOut := ScrewInTube); END_IF;
(* Rung 1 *)
_e2(CLK := iFeedSOL);
IF _e2.Q THEN
    ScrewInClamp := ScrewInTube;
    ScrewInTube := int#0;
END_IF;
(* Rung 2 *)
oCheckError := ScrewInClamp = int#0;
(* Rung 3 *)
IF iResetPB THEN ScrewInClamp := int#1; END_IF;
END_FUNCTION_BLOCK

FUNCTION_BLOCK FeedScrewFlow
VAR
    TON_PON : TON;
    PowerOn : BOOL;
    TON_PowerOn : TON;
    Idle : BOOL;
    FeedStart : BOOL;
    Feeding : BOOL;
    Feeded : BOOL;
    FeedAgain : BOOL;
    FeedFinish : BOOL;
    ClearCount : BOOL;
    match : BOOL;  (* 符合設定數量 *)
    less : BOOL;  (* 數量不足 *)
    TON_S8110FeedAgain : TON;
END_VAR
VAR_INPUT
    ENABLE : BOOL;
    bStartFlag : BOOL;
    bResetFlag : BOOL;
    bFeedSOL : BOOL;
    bFeedError : BOOL;
    iQuantitySV : INT;
END_VAR
VAR_OUTPUT
    bFeedStartFlag : BOOL;
END_VAR
VAR_IN_OUT
    iCounter : INT;
END_VAR
VAR
    _e1 : R_TRIG;
    _e2 : R_TRIG;
END_VAR
(* ladder, written here as Structured Text *)

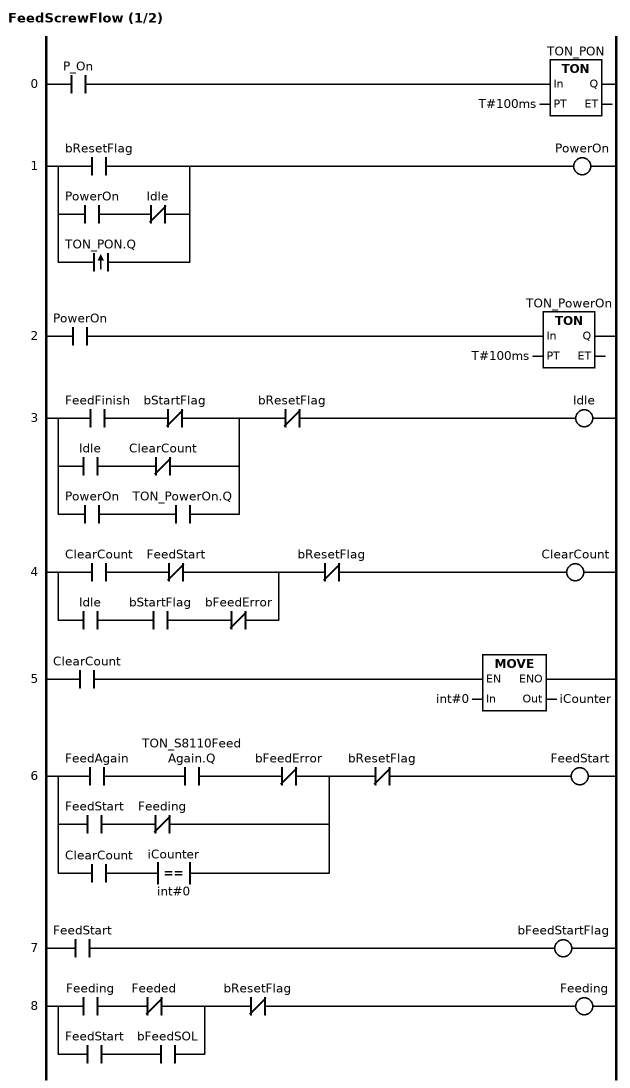
(* Rung 0 *)
TON_PON(In := P_On, PT := T#100ms);
(* Rung 1 *)
_e1(CLK := TON_PON.Q);
PowerOn := bResetFlag OR (PowerOn AND NOT Idle) OR _e1.Q;
(* Rung 2 *)
TON_PowerOn(In := PowerOn, PT := T#100ms);
(* Rung 3 *)
Idle := ((FeedFinish AND NOT bStartFlag) OR (Idle AND NOT ClearCount) OR (PowerOn AND TON_PowerOn.Q)) AND NOT bResetFlag;
(* Rung 4 *)
ClearCount := ((ClearCount AND NOT FeedStart) OR (Idle AND bStartFlag AND NOT bFeedError)) AND NOT bResetFlag;
(* Rung 5 *)
IF ClearCount THEN iCounter := int#0; END_IF;
(* Rung 6 *)
FeedStart := ((FeedAgain AND TON_S8110FeedAgain.Q AND NOT bFeedError) OR (FeedStart AND NOT Feeding) OR (ClearCount AND (iCounter = int#0))) AND NOT bResetFlag;
(* Rung 7 *)
bFeedStartFlag := FeedStart;
(* Rung 8 *)
Feeding := ((Feeding AND NOT Feeded) OR (FeedStart AND bFeedSOL)) AND NOT bResetFlag;

